  MoveL 8802 to (-24.03, 35.21, 125.68) mm, rotated rx 180 ry 0 rz 180 deg; joints [-34.794, -28.488, 103.329, 69.378, 37.567, -64.603]
  MoveL 8803 to (-24.03, 35.21, 125.68) mm, rotated rx 180 ry 0 rz 180 deg; joints [-34.794, -28.488, 103.329, 69.378, 37.567, -64.603]
  Call Extruder(470.65922)
  MoveL 8804 to (-23.64, 35.16, 125.68) mm, rotated rx 180 ry 0 rz 180 deg; joints [-34.738, -28.447, 103.308, 69.362, 37.51, -64.602]
  MoveL 8805 to (-23.64, 35.16, 125.68) mm, rotated rx 180 ry 0 rz 180 deg; joints [-34.738, -28.447, 103.308, 69.362, 37.51, -64.602]
  Call Extruder(470.90490)
  MoveL 8806 to (-23.15, 35.11, 125.68) mm, rotated rx 180 ry 0 rz 180 deg; joints [-34.671, -28.395, 103.28, 69.345, 37.441, -64.602]
  MoveL 8807 to (-23.15, 35.11, 125.68) mm, rotated rx 180 ry 0 rz 180 deg; joints [-34.671, -28.395, 103.28, 69.345, 37.441, -64.602]
  Call Extruder(471.19963)
  MoveL 8808 to (-22.56, 35.07, 125.68) mm, rotated rx 180 ry 0 rz 180 deg; joints [-34.592, -28.331, 103.247, 69.326, 37.359, -64.604]
  MoveL 8809 to (-22.56, 35.07, 125.68) mm, rotated rx 180 ry 0 rz 180 deg; joints [-34.592, -28.331, 103.247, 69.326, 37.359, -64.604]
  Call Extruder(471.49303)
  MoveL 8810 to (-21.97, 35.02, 125.68) mm, rotated rx -180 ry 0 rz 180 deg; joints [-34.512, -28.267, 103.213, 69.307, 37.276, -64.606]
  MoveL 8811 to (-21.97, 35.02, 125.68) mm, rotated rx -180 ry 0 rz 180 deg; joints [-34.512, -28.267, 103.213, 69.307, 37.276, -64.606]
  Call Extruder(471.92636)
  MoveL 8812 to (-21.1, 34.98, 125.68) mm, rotated rx 180 ry 0 rz -180 deg; joints [-34.399, -28.17, 103.162, 69.282, 37.158, -64.612]
  MoveL 8813 to (-21.1, 34.98, 125.68) mm, rotated rx 180 ry 0 rz -180 deg; joints [-34.399, -28.17, 103.162, 69.282, 37.158, -64.612]
  Call Extruder(472.49852)
  MoveL 8814 to (-19.94, 34.93, 125.68) mm, rotated rx 180 ry 0 rz 180 deg; joints [-34.253, -28.04, 103.092, 69.254, 37.004, -64.624]
  MoveL 8815 to (-19.94, 34.93, 125.68) mm, rotated rx 180 ry 0 rz 180 deg; joints [-34.253, -28.04, 103.092, 69.254, 37.004, -64.624]
  Call Extruder(472.92635)
  MoveL 8816 to (-19.06, 34.91, 125.68) mm, rotated rx -180 ry 0 rz 180 deg; joints [-34.146, -27.941, 103.039, 69.235, 36.891, -64.635]
  Call Extruder(589.57504)
  MoveL 8817 to (219.06, 34.91, 125.68) mm, rotated rx 180 ry 0 rz 180 deg; joints [-18.248, 4.075, 77.332, 65.623, 20.108, -64.241]
  MoveL 8818 to (219.06, 34.91, 125.68) mm, rotated rx 180 ry 0 rz 180 deg; joints [-18.248, 4.075, 77.332, 65.623, 20.108, -64.241]
  Call Extruder(590.29061)
  MoveL 8819 to (220.52, 34.95, 125.68) mm, rotated rx -180 ry 0 rz 180 deg; joints [-18.199, 4.301, 77.091, 65.523, 20.07, -64.141]
  MoveL 8820 to (220.52, 34.95, 125.68) mm, rotated rx -180 ry 0 rz 180 deg; joints [-18.199, 4.301, 77.091, 65.523, 20.07, -64.141]
  Call Extruder(590.86535)
  MoveL 8821 to (221.68, 35, 125.68) mm, rotated rx 180 ry 0 rz 180 deg; joints [-18.162, 4.483, 76.896, 65.442, 20.042, -64.062]
  MoveL 8822 to (221.68, 35, 125.68) mm, rotated rx 180 ry 0 rz 180 deg; joints [-18.162, 4.483, 76.896, 65.442, 20.042, -64.062]
  Call Extruder(591.15874)
  MoveL 8823 to (222.27, 35.04, 125.68) mm, rotated rx -180 ry 0 rz 180 deg; joints [-18.146, 4.576, 76.796, 65.404, 20.03, -64.024]
  MoveL 8824 to (222.27, 35.04, 125.68) mm, rotated rx -180 ry 0 rz 180 deg; joints [-18.146, 4.576, 76.796, 65.404, 20.03, -64.024]
  Call Extruder(591.45347)
  MoveL 8825 to (222.86, 35.09, 125.68) mm, rotated rx 180 ry 0 rz 180 deg; joints [-18.13, 4.669, 76.695, 65.366, 20.018, -63.986]
  MoveL 8826 to (222.86, 35.09, 125.68) mm, rotated rx 180 ry 0 rz 180 deg; joints [-18.13, 4.669, 76.695, 65.366, 20.018, -63.986]
  Call Extruder(591.74952)
  MoveL 8827 to (223.45, 35.14, 125.68) mm, rotated rx 180 ry 0 rz -180 deg; joints [-18.113, 4.763, 76.594, 65.327, 20.007, -63.947]
  MoveL 8828 to (223.45, 35.14, 125.68) mm, rotated rx 180 ry 0 rz -180 deg; joints [-18.113, 4.763, 76.594, 65.327, 20.007, -63.947]
  Call Extruder(591.94580)
  MoveL 8829 to (223.84, 35.18, 125.68) mm, rotated rx -180 ry 0 rz 180 deg; joints [-18.104, 4.825, 76.527, 65.303, 20.001, -63.923]
  MoveL 8830 to (223.84, 35.18, 125.68) mm, rotated rx -180 ry 0 rz 180 deg; joints [-18.104, 4.825, 76.527, 65.303, 20.001, -63.923]
  Call Extruder(592.14294)
  MoveL 8831 to (224.22, 35.23, 125.68) mm, rotated rx -180 ry 0 rz 180 deg; joints [-18.095, 4.888, 76.46, 65.279, 19.995, -63.899]
  MoveL 8832 to (224.22, 35.23, 125.68) mm, rotated rx -180 ry 0 rz 180 deg; joints [-18.095, 4.888, 76.46, 65.279, 19.995, -63.899]
  Call Extruder(592.34095)
  MoveL 8833 to (224.61, 35.27, 125.68) mm, rotated rx 180 ry 0 rz 180 deg; joints [-18.087, 4.95, 76.393, 65.255, 19.989, -63.875]
  MoveL 8834 to (224.61, 35.27, 125.68) mm, rotated rx 180 ry 0 rz 180 deg; joints [-18.087, 4.95, 76.393, 65.255, 19.989, -63.875]
  Call Extruder(592.53982)
  MoveL 8835 to (225, 35.32, 125.68) mm, rotated rx 180 ry 0 rz 180 deg; joints [-18.078, 5.012, 76.325, 65.231, 19.983, -63.85]
  MoveL 8836 to (225, 35.32, 125.68) mm, rotated rx 180 ry 0 rz 180 deg; joints [-18.078, 5.012, 76.325, 65.231, 19.983, -63.85]
  Call Extruder(592.71890)
  MoveL 8837 to (225.34, 35.37, 125.68) mm, rotated rx 180 ry 0 rz 180 deg; joints [-18.07, 5.068, 76.264, 65.21, 19.979, -63.829]
  MoveL 8838 to (225.34, 35.37, 125.68) mm, rotated rx 180 ry 0 rz 180 deg; joints [-18.07, 5.068, 76.264, 65.21, 19.979, -63.829]
  Call Extruder(592.87809)
  MoveL 8839 to (225.65, 35.42, 125.68) mm, rotated rx 180 ry 0 rz 180 deg; joints [-18.065, 5.118, 76.21, 65.192, 19.975, -63.811]
  MoveL 8840 to (225.65, 35.42, 125.68) mm, rotated rx 180 ry 0 rz 180 deg; joints [-18.065, 5.118, 76.21, 65.192, 19.975, -63.811]
  Call Extruder(593.03800)
  MoveL 8841 to (225.96, 35.46, 125.68) mm, rotated rx 180 ry 0 rz 180 deg; joints [-18.059, 5.168, 76.156, 65.174, 19.972, -63.793]
  MoveL 8842 to (225.96, 35.46, 125.68) mm, rotated rx 180 ry 0 rz 180 deg; joints [-18.059, 5.168, 76.156, 65.174, 19.972, -63.793]
  Call Extruder(593.19864)
  MoveL 8843 to (226.26, 35.51, 125.68) mm, rotated rx 180 ry 0 rz 180 deg; joints [-18.054, 5.218, 76.102, 65.156, 19.969, -63.775]
  MoveL 8844 to (226.26, 35.51, 125.68) mm, rotated rx 180 ry 0 rz 180 deg; joints [-18.054, 5.218, 76.102, 65.156, 19.969, -63.775]
  Call Extruder(593.36001)
  MoveL 8845 to (226.57, 35.56, 125.68) mm, rotated rx -180 ry 0 rz 180 deg; joints [-18.048, 5.268, 76.048, 65.138, 19.966, -63.757]
  MoveL 8846 to (226.57, 35.56, 125.68) mm, rotated rx -180 ry 0 rz 180 deg; joints [-18.048, 5.268, 76.048, 65.138, 19.966, -63.757]
  Call Extruder(593.52210)
  MoveL 8847 to (226.87, 35.61, 125.68) mm, rotated rx 180 ry 0 rz -180 deg; joints [-18.042, 5.318, 75.993, 65.12, 19.962, -63.738]
  MoveL 8848 to (226.87, 35.61, 125.68) mm, rotated rx 180 ry 0 rz -180 deg; joints [-18.042, 5.318, 75.993, 65.12, 19.962, -63.738]
  Call Extruder(593.67030)
  MoveL 8849 to (227.15, 35.66, 125.68) mm, rotated rx 180 ry 0 rz 180 deg; joints [-18.038, 5.364, 75.944, 65.104, 19.96, -63.722]
  MoveL 8850 to (227.15, 35.66, 125.68) mm, rotated rx 180 ry 0 rz 180 deg; joints [-18.038, 5.364, 75.944, 65.104, 19.96, -63.722]
  Call Extruder(593.80453)
  MoveL 8851 to (227.4, 35.71, 125.68) mm, rotated rx 180 ry 0 rz 180 deg; joints [-18.034, 5.405, 75.899, 65.091, 19.958, -63.708]
  MoveL 8852 to (227.4, 35.71, 125.68) mm, rotated rx 180 ry 0 rz 180 deg; joints [-18.034, 5.405, 75.899, 65.091, 19.958, -63.708]
  Call Extruder(593.93938)
  MoveL 8853 to (227.65, 35.76, 125.68) mm, rotated rx 180 ry 0 rz 180 deg; joints [-18.031, 5.446, 75.854, 65.077, 19.957, -63.694]
  MoveL 8854 to (227.65, 35.76, 125.68) mm, rotated rx 180 ry 0 rz 180 deg; joints [-18.031, 5.446, 75.854, 65.077, 19.957, -63.694]
  Call Extruder(594.07483)
  MoveL 8855 to (227.9, 35.81, 125.68) mm, rotated rx 180 ry 0 rz 180 deg; joints [-18.027, 5.488, 75.809, 65.063, 19.955, -63.68]
  MoveL 8856 to (227.9, 35.81, 125.68) mm, rotated rx 180 ry 0 rz 180 deg; joints [-18.027, 5.488, 75.809, 65.063, 19.955, -63.68]
  Call Extruder(594.21089)
  MoveL 8857 to (228.15, 35.86, 125.68) mm, rotated rx 180 ry 0 rz -180 deg; joints [-18.024, 5.529, 75.764, 65.049, 19.954, -63.666]
  MoveL 8858 to (228.15, 35.86, 125.68) mm, rotated rx 180 ry 0 rz -180 deg; joints [-18.024, 5.529, 75.764, 65.049, 19.954, -63.666]
  Call Extruder(594.34757)
  MoveL 8859 to (228.4, 35.91, 125.68) mm, rotated rx 180 ry 0 rz 180 deg; joints [-18.02, 5.57, 75.719, 65.035, 19.952, -63.651]
  MoveL 8860 to (228.4, 35.91, 125.68) mm, rotated rx 180 ry 0 rz 180 deg; joints [-18.02, 5.57, 75.719, 65.035, 19.952, -63.651]
  Call Extruder(594.48485)
  MoveL 8861 to (228.65, 35.96, 125.68) mm, rotated rx 180 ry 0 rz 180 deg; joints [-18.017, 5.612, 75.673, 65.021, 19.951, -63.637]
  MoveL 8862 to (228.65, 35.96, 125.68) mm, rotated rx 180 ry 0 rz 180 deg; joints [-18.017, 5.612, 75.673, 65.021, 19.951, -63.637]
  Call Extruder(594.61052)
  MoveL 8863 to (228.87, 36, 125.68) mm, rotated rx 180 ry 0 rz 180 deg; joints [-18.014, 5.649, 75.632, 65.009, 19.95, -63.624]
  MoveL 8864 to (228.87, 36, 125.68) mm, rotated rx 180 ry 0 rz 180 deg; joints [-18.014, 5.649, 75.632, 65.009, 19.95, -63.624]
  Call Extruder(594.72447)
  MoveL 8865 to (229.08, 36.05, 125.68) mm, rotated rx -180 ry 0 rz -180 deg; joints [-18.012, 5.684, 75.595, 64.998, 19.949, -63.613]
  MoveL 8866 to (229.08, 36.05, 125.68) mm, rotated rx -180 ry 0 rz -180 deg; joints [-18.012, 5.684, 75.595, 64.998, 19.949, -63.613]
  Call Extruder(594.83887)
  MoveL 8867 to (229.28, 36.09, 125.68) mm, rotated rx 180 ry 0 rz 180 deg; joints [-18.009, 5.718, 75.558, 64.987, 19.948, -63.602]
  MoveL 8868 to (229.28, 36.09, 125.68) mm, rotated rx 180 ry 0 rz 180 deg; joints [-18.009, 5.718, 75.558, 64.987, 19.948, -63.602]
  Call Extruder(594.95372)
  MoveL 8869 to (229.48, 36.14, 125.68) mm, rotated rx -180 ry 0 rz 180 deg; joints [-18.007, 5.752, 75.52, 64.976, 19.947, -63.59]
  MoveL 8870 to (229.48, 36.14, 125.68) mm, rotated rx -180 ry 0 rz 180 deg; joints [-18.007, 5.752, 75.52, 64.976, 19.947, -63.59]
  Call Extruder(595.06902)
  MoveL 8871 to (229.69, 36.18, 125.68) mm, rotated rx 180 ry 0 rz 180 deg; joints [-18.005, 5.786, 75.483, 64.965, 19.947, -63.579]
  MoveL 8872 to (229.69, 36.18, 125.68) mm, rotated rx 180 ry 0 rz 180 deg; joints [-18.005, 5.786, 75.483, 64.965, 19.947, -63.579]
  Call Extruder(595.20041)
  MoveL 8873 to (229.92, 36.25, 125.68) mm, rotated rx 180 ry 0 rz -180 deg; joints [-18.004, 5.825, 75.44, 64.954, 19.947, -63.568]
  MoveL 8874 to (229.92, 36.25, 125.68) mm, rotated rx 180 ry 0 rz -180 deg; joints [-18.004, 5.825, 75.44, 64.954, 19.947, -63.568]
  Call Extruder(595.31352)
  MoveL 8875 to (230.11, 36.31, 125.68) mm, rotated rx 180 ry 0 rz 180 deg; joints [-18.003, 5.858, 75.403, 64.945, 19.948, -63.558]
  MoveL 8876 to (230.11, 36.31, 125.68) mm, rotated rx 180 ry 0 rz 180 deg; joints [-18.003, 5.858, 75.403, 64.945, 19.948, -63.558]
  Call Extruder(595.42707)
  MoveL 8877 to (230.31, 36.37, 125.68) mm, rotated rx 180 ry 0 rz 180 deg; joints [-18.003, 5.892, 75.367, 64.937, 19.949, -63.549]
  MoveL 8878 to (230.31, 36.37, 125.68) mm, rotated rx 180 ry 0 rz 180 deg; joints [-18.003, 5.892, 75.367, 64.937, 19.949, -63.549]
  Call Extruder(595.54106)
  MoveL 8879 to (230.5, 36.43, 125.68) mm, rotated rx 180 ry 0 rz -180 deg; joints [-18.002, 5.925, 75.33, 64.928, 19.95, -63.54]
  MoveL 8880 to (230.5, 36.43, 125.68) mm, rotated rx 180 ry 0 rz -180 deg; joints [-18.002, 5.925, 75.33, 64.928, 19.95, -63.54]
  Call Extruder(595.65549)
  MoveL 8881 to (230.69, 36.49, 125.68) mm, rotated rx 180 ry 0 rz 180 deg; joints [-18.002, 5.959, 75.293, 64.92, 19.951, -63.531]
  MoveL 8882 to (230.69, 36.49, 125.68) mm, rotated rx 180 ry 0 rz 180 deg; joints [-18.002, 5.959, 75.293, 64.92, 19.951, -63.531]
  Call Extruder(595.76739)
  MoveL 8883 to (230.88, 36.55, 125.68) mm, rotated rx 180 ry 0 rz 180 deg; joints [-18.002, 5.991, 75.257, 64.912, 19.953, -63.523]
  MoveL 8884 to (230.88, 36.55, 125.68) mm, rotated rx 180 ry 0 rz 180 deg; joints [-18.002, 5.991, 75.257, 64.912, 19.953, -63.523]
  Call Extruder(595.87973)
  MoveL 8885 to (231.07, 36.61, 125.68) mm, rotated rx 180 ry 0 rz 180 deg; joints [-18.002, 6.024, 75.222, 64.903, 19.954, -63.514]
  MoveL 8886 to (231.07, 36.61, 125.68) mm, rotated rx 180 ry 0 rz 180 deg; joints [-18.002, 6.024, 75.222, 64.903, 19.954, -63.514]
  Call Extruder(595.99252)
  MoveL 8887 to (231.26, 36.67, 125.68) mm, rotated rx 180 ry 0 rz 180 deg; joints [-18.002, 6.057, 75.186, 64.895, 19.956, -63.506]
  MoveL 8888 to (231.26, 36.67, 125.68) mm, rotated rx 180 ry 0 rz 180 deg; joints [-18.002, 6.057, 75.186, 64.895, 19.956, -63.506]
  Call Extruder(596.10575)
  MoveL 8889 to (231.45, 36.73, 125.68) mm, rotated rx 180 ry 0 rz 180 deg; joints [-18.002, 6.089, 75.15, 64.887, 19.957, -63.497]
  MoveL 8890 to (231.45, 36.73, 125.68) mm, rotated rx 180 ry 0 rz 180 deg; joints [-18.002, 6.089, 75.15, 64.887, 19.957, -63.497]
  Call Extruder(596.21943)
  MoveL 8891 to (231.64, 36.79, 125.68) mm, rotated rx 180 ry 0 rz 180 deg; joints [-18.002, 6.122, 75.114, 64.879, 19.958, -63.488]
  MoveL 8892 to (231.64, 36.79, 125.68) mm, rotated rx 180 ry 0 rz 180 deg; joints [-18.002, 6.122, 75.114, 64.879, 19.958, -63.488]
  Call Extruder(596.40139)
  MoveL 8893 to (231.93, 36.91, 125.68) mm, rotated rx 180 ry 0 rz 180 deg; joints [-18.005, 6.174, 75.057, 64.87, 19.963, -63.478]
  MoveL 8894 to (231.93, 36.91, 125.68) mm, rotated rx 180 ry 0 rz 180 deg; joints [-18.005, 6.174, 75.057, 64.87, 19.963, -63.478]
  Call Extruder(596.58411)
  MoveL 8895 to (232.22, 37.04, 125.68) mm, rotated rx 180 ry 0 rz -180 deg; joints [-18.008, 6.226, 74.999, 64.86, 19.968, -63.467]
  MoveL 8896 to (232.22, 37.04, 125.68) mm, rotated rx 180 ry 0 rz -180 deg; joints [-18.008, 6.226, 74.999, 64.86, 19.968, -63.467]
  Call Extruder(596.75452)
  MoveL 8897 to (232.49, 37.15, 125.68) mm, rotated rx 180 ry 0 rz 180 deg; joints [-18.011, 6.274, 74.946, 64.852, 19.973, -63.458]
  MoveL 8898 to (232.49, 37.15, 125.68) mm, rotated rx 180 ry 0 rz 180 deg; joints [-18.011, 6.274, 74.946, 64.852, 19.973, -63.458]
  Call Extruder(596.91252)
  MoveL 8899 to (232.74, 37.26, 125.68) mm, rotated rx -180 ry 0 rz -180 deg; joints [-18.013, 6.319, 74.897, 64.844, 19.977, -63.449]
  MoveL 8900 to (232.74, 37.26, 125.68) mm, rotated rx -180 ry 0 rz -180 deg; joints [-18.013, 6.319, 74.897, 64.844, 19.977, -63.449]
  Call Extruder(597.07112)
  MoveL 8901 to (232.99, 37.36, 125.68) mm, rotated rx -180 ry 0 rz 180 deg; joints [-18.016, 6.363, 74.848, 64.836, 19.982, -63.44]
  MoveL 8902 to (232.99, 37.36, 125.68) mm, rotated rx -180 ry 0 rz 180 deg; joints [-18.016, 6.363, 74.848, 64.836, 19.982, -63.44]
  Call Extruder(597.27729)
  MoveL 8903 to (233.29, 37.54, 125.68) mm, rotated rx 180 ry 0 rz 180 deg; joints [-18.024, 6.42, 74.785, 64.832, 19.991, -63.434]
  MoveL 8904 to (233.29, 37.54, 125.68) mm, rotated rx 180 ry 0 rz 180 deg; joints [-18.024, 6.42, 74.785, 64.832, 19.991, -63.434]
  Call Extruder(597.48423)
  MoveL 8905 to (233.6, 37.71, 125.68) mm, rotated rx 180 ry 0 rz 180 deg; joints [-18.033, 6.477, 74.722, 64.828, 20.001, -63.429]
  MoveL 8906 to (233.6, 37.71, 125.68) mm, rotated rx 180 ry 0 rz 180 deg; joints [-18.033, 6.477, 74.722, 64.828, 20.001, -63.429]
  Call Extruder(597.69196)
  MoveL 8907 to (233.9, 37.89, 125.68) mm, rotated rx -180 ry 0 rz -180 deg; joints [-18.041, 6.534, 74.66, 64.823, 20.011, -63.423]
  MoveL 8908 to (233.9, 37.89, 125.68) mm, rotated rx -180 ry 0 rz -180 deg; joints [-18.041, 6.534, 74.66, 64.823, 20.011, -63.423]
  Call Extruder(597.90046)
  MoveL 8909 to (234.21, 38.07, 125.68) mm, rotated rx 180 ry 0 rz 180 deg; joints [-18.049, 6.59, 74.597, 64.819, 20.021, -63.417]
  MoveL 8910 to (234.21, 38.07, 125.68) mm, rotated rx 180 ry 0 rz 180 deg; joints [-18.049, 6.59, 74.597, 64.819, 20.021, -63.417]
  Call Extruder(598.08001)
  MoveL 8911 to (234.45, 38.24, 125.68) mm, rotated rx 180 ry 0 rz 180 deg; joints [-18.06, 6.638, 74.544, 64.82, 20.033, -63.416]
  MoveL 8912 to (234.45, 38.24, 125.68) mm, rotated rx 180 ry 0 rz 180 deg; joints [-18.06, 6.638, 74.544, 64.82, 20.033, -63.416]
  Call Extruder(598.41342)
  MoveL 8913 to (234.9, 38.57, 125.68) mm, rotated rx 180 ry 0 rz 180 deg; joints [-18.079, 6.726, 74.446, 64.821, 20.055, -63.414]
  MoveL 8914 to (234.9, 38.57, 125.68) mm, rotated rx 180 ry 0 rz 180 deg; joints [-18.079, 6.726, 74.446, 64.821, 20.055, -63.414]
  Call Extruder(598.74802)
  MoveL 8915 to (235.35, 38.9, 125.68) mm, rotated rx 180 ry 0 rz 180 deg; joints [-18.099, 6.814, 74.348, 64.823, 20.076, -63.412]
  Call Extruder(599.57597)
  MoveL 8916 to (236.39, 39.81, 125.68) mm, rotated rx 180 ry 0 rz -180 deg; joints [-18.16, 7.025, 74.114, 64.844, 20.142, -63.425]
  Call Extruder(600.40391)
  MoveL 8917 to (237.3, 40.85, 125.68) mm, rotated rx 180 ry 0 rz -180 deg; joints [-18.24, 7.223, 73.892, 64.889, 20.222, -63.46]
  Call Extruder(600.57121)
  MoveL 8918 to (237.47, 41.07, 125.68) mm, rotated rx -180 ry 0 rz 180 deg; joints [-18.258, 7.26, 73.85, 64.902, 20.241, -63.471]
  MoveL 8919 to (237.47, 41.07, 125.68) mm, rotated rx -180 ry 0 rz 180 deg; joints [-18.258, 7.26, 73.85, 64.902, 20.241, -63.471]
  Call Extruder(600.90463)
  MoveL 8920 to (237.8, 41.52, 125.68) mm, rotated rx 180 ry 0 rz 180 deg; joints [-18.295, 7.336, 73.766, 64.927, 20.277, -63.491]
  MoveL 8921 to (237.8, 41.52, 125.68) mm, rotated rx 180 ry 0 rz 180 deg; joints [-18.295, 7.336, 73.766, 64.927, 20.277, -63.491]
  Call Extruder(601.23686)
  MoveL 8922 to (238.12, 41.98, 125.68) mm, rotated rx -180 ry 0 rz 180 deg; joints [-18.332, 7.412, 73.681, 64.952, 20.314, -63.512]
  MoveL 8923 to (238.12, 41.98, 125.68) mm, rotated rx -180 ry 0 rz 180 deg; joints [-18.332, 7.412, 73.681, 64.952, 20.314, -63.512]
  Call Extruder(601.35455)
  MoveL 8924 to (238.22, 42.15, 125.68) mm, rotated rx 180 ry 0 rz 180 deg; joints [-18.346, 7.436, 73.653, 64.963, 20.329, -63.522]
  MoveL 8925 to (238.22, 42.15, 125.68) mm, rotated rx 180 ry 0 rz 180 deg; joints [-18.346, 7.436, 73.653, 64.963, 20.329, -63.522]
  Call Extruder(601.56228)
  MoveL 8926 to (238.4, 42.45, 125.68) mm, rotated rx 180 ry 0 rz 180 deg; joints [-18.373, 7.48, 73.604, 64.984, 20.354, -63.539]
  MoveL 8927 to (238.4, 42.45, 125.68) mm, rotated rx 180 ry 0 rz 180 deg; joints [-18.373, 7.48, 73.604, 64.984, 20.354, -63.539]
  Call Extruder(601.76922)
  MoveL 8928 to (238.57, 42.75, 125.68) mm, rotated rx 180 ry 0 rz -180 deg; joints [-18.399, 7.524, 73.555, 65.004, 20.38, -63.557]
  MoveL 8929 to (238.57, 42.75, 125.68) mm, rotated rx 180 ry 0 rz -180 deg; joints [-18.399, 7.524, 73.555, 65.004, 20.38, -63.557]
  Call Extruder(601.97539)
  MoveL 8930 to (238.75, 43.06, 125.68) mm, rotated rx 180 ry 0 rz 180 deg; joints [-18.425, 7.568, 73.506, 65.025, 20.406, -63.574]
  MoveL 8931 to (238.75, 43.06, 125.68) mm, rotated rx 180 ry 0 rz 180 deg; joints [-18.425, 7.568, 73.506, 65.025, 20.406, -63.574]
  Call Extruder(602.15708)
  MoveL 8932 to (238.89, 43.34, 125.68) mm, rotated rx 180 ry 0 rz 180 deg; joints [-18.45, 7.605, 73.464, 65.045, 20.43, -63.591]
  MoveL 8933 to (238.89, 43.34, 125.68) mm, rotated rx 180 ry 0 rz 180 deg; joints [-18.45, 7.605, 73.464, 65.045, 20.43, -63.591]
  Call Extruder(602.31509)
  MoveL 8934 to (239, 43.58, 125.68) mm, rotated rx 180 ry 0 rz 180 deg; joints [-18.472, 7.635, 73.43, 65.064, 20.452, -63.608]
  MoveL 8935 to (239, 43.58, 125.68) mm, rotated rx 180 ry 0 rz 180 deg; joints [-18.472, 7.635, 73.43, 65.064, 20.452, -63.608]
  Call Extruder(602.47250)
  MoveL 8936 to (239.11, 43.83, 125.68) mm, rotated rx 180 ry 0 rz 180 deg; joints [-18.495, 7.665, 73.396, 65.084, 20.474, -63.626]
  MoveL 8937 to (239.11, 43.83, 125.68) mm, rotated rx 180 ry 0 rz 180 deg; joints [-18.495, 7.665, 73.396, 65.084, 20.474, -63.626]
  Call Extruder(602.65521)
  MoveL 8938 to (239.23, 44.13, 125.68) mm, rotated rx 180 ry 0 rz 180 deg; joints [-18.522, 7.7, 73.357, 65.107, 20.5, -63.646]
  MoveL 8939 to (239.23, 44.13, 125.68) mm, rotated rx 180 ry 0 rz 180 deg; joints [-18.522, 7.7, 73.357, 65.107, 20.5, -63.646]
  Call Extruder(602.83717)
  MoveL 8940 to (239.35, 44.42, 125.68) mm, rotated rx 180 ry 0 rz 180 deg; joints [-18.549, 7.734, 73.318, 65.131, 20.526, -63.667]
  MoveL 8941 to (239.35, 44.42, 125.68) mm, rotated rx 180 ry 0 rz 180 deg; joints [-18.549, 7.734, 73.318, 65.131, 20.526, -63.667]
  Call Extruder(602.98450)
  MoveL 8942 to (239.44, 44.66, 125.68) mm, rotated rx 180 ry 0 rz -180 deg; joints [-18.571, 7.762, 73.287, 65.15, 20.547, -63.684]
  MoveL 8943 to (239.44, 44.66, 125.68) mm, rotated rx 180 ry 0 rz -180 deg; joints [-18.571, 7.762, 73.287, 65.15, 20.547, -63.684]
  Call Extruder(603.09774)
  MoveL 8944 to (239.5, 44.85, 125.68) mm, rotated rx -180 ry 0 rz 180 deg; joints [-18.589, 7.782, 73.265, 65.167, 20.564, -63.699]
  MoveL 8945 to (239.5, 44.85, 125.68) mm, rotated rx -180 ry 0 rz 180 deg; joints [-18.589, 7.782, 73.265, 65.167, 20.564, -63.699]
  Call Extruder(603.21053)
  MoveL 8946 to (239.56, 45.03, 125.68) mm, rotated rx 180 ry 0 rz 180 deg; joints [-18.607, 7.801, 73.242, 65.183, 20.581, -63.713]
  MoveL 8947 to (239.56, 45.03, 125.68) mm, rotated rx 180 ry 0 rz 180 deg; joints [-18.607, 7.801, 73.242, 65.183, 20.581, -63.713]
  Call Extruder(603.32287)
  MoveL 8948 to (239.62, 45.22, 125.68) mm, rotated rx 180 ry 0 rz 180 deg; joints [-18.625, 7.821, 73.22, 65.2, 20.598, -63.728]
  MoveL 8949 to (239.62, 45.22, 125.68) mm, rotated rx 180 ry 0 rz 180 deg; joints [-18.625, 7.821, 73.22, 65.2, 20.598, -63.728]
  Call Extruder(603.43477)
  MoveL 8950 to (239.68, 45.41, 125.68) mm, rotated rx 180 ry 0 rz -180 deg; joints [-18.642, 7.841, 73.198, 65.216, 20.615, -63.742]
  MoveL 8951 to (239.68, 45.41, 125.68) mm, rotated rx 180 ry 0 rz -180 deg; joints [-18.642, 7.841, 73.198, 65.216, 20.615, -63.742]
  Call Extruder(603.55618)
  MoveL 8952 to (239.75, 45.62, 125.68) mm, rotated rx 180 ry 0 rz -180 deg; joints [-18.662, 7.862, 73.174, 65.234, 20.634, -63.758]
  MoveL 8953 to (239.75, 45.62, 125.68) mm, rotated rx 180 ry 0 rz -180 deg; joints [-18.662, 7.862, 73.174, 65.234, 20.634, -63.758]
  Call Extruder(603.68697)
  MoveL 8954 to (239.81, 45.84, 125.68) mm, rotated rx 180 ry 0 rz 180 deg; joints [-18.683, 7.885, 73.148, 65.253, 20.654, -63.775]
  MoveL 8955 to (239.81, 45.84, 125.68) mm, rotated rx 180 ry 0 rz 180 deg; joints [-18.683, 7.885, 73.148, 65.253, 20.654, -63.775]
  Call Extruder(603.81719)
  MoveL 8956 to (239.88, 46.06, 125.68) mm, rotated rx 180 ry 0 rz -180 deg; joints [-18.705, 7.908, 73.122, 65.273, 20.675, -63.793]
  MoveL 8957 to (239.88, 46.06, 125.68) mm, rotated rx 180 ry 0 rz -180 deg; joints [-18.705, 7.908, 73.122, 65.273, 20.675, -63.793]
  Call Extruder(603.94685)
  MoveL 8958 to (239.95, 46.29, 125.68) mm, rotated rx 180 ry 0 rz 180 deg; joints [-18.726, 7.93, 73.096, 65.292, 20.695, -63.81]
  MoveL 8959 to (239.95, 46.29, 125.68) mm, rotated rx 180 ry 0 rz 180 deg; joints [-18.726, 7.93, 73.096, 65.292, 20.695, -63.81]
  Call Extruder(604.07595)
  MoveL 8960 to (240.02, 46.51, 125.68) mm, rotated rx 180 ry 0 rz -180 deg; joints [-18.747, 7.953, 73.071, 65.312, 20.715, -63.827]
  MoveL 8961 to (240.02, 46.51, 125.68) mm, rotated rx 180 ry 0 rz -180 deg; joints [-18.747, 7.953, 73.071, 65.312, 20.715, -63.827]
  Call Extruder(604.19100)
  MoveL 8962 to (240.06, 46.72, 125.68) mm, rotated rx 180 ry 0 rz 180 deg; joints [-18.767, 7.971, 73.05, 65.331, 20.734, -63.844]
  MoveL 8963 to (240.06, 46.72, 125.68) mm, rotated rx 180 ry 0 rz 180 deg; joints [-18.767, 7.971, 73.05, 65.331, 20.734, -63.844]
  Call Extruder(604.30560)
  MoveL 8964 to (240.11, 46.92, 125.68) mm, rotated rx 180 ry 0 rz 180 deg; joints [-18.787, 7.989, 73.03, 65.35, 20.753, -63.862]
  MoveL 8965 to (240.11, 46.92, 125.68) mm, rotated rx 180 ry 0 rz 180 deg; joints [-18.787, 7.989, 73.03, 65.35, 20.753, -63.862]
  Call Extruder(604.41975)
  MoveL 8966 to (240.15, 47.12, 125.68) mm, rotated rx 180 ry 0 rz 180 deg; joints [-18.807, 8.007, 73.009, 65.37, 20.772, -63.879]
  MoveL 8967 to (240.15, 47.12, 125.68) mm, rotated rx 180 ry 0 rz 180 deg; joints [-18.807, 8.007, 73.009, 65.37, 20.772, -63.879]
  Call Extruder(604.53345)
  MoveL 8968 to (240.2, 47.33, 125.68) mm, rotated rx -180 ry 0 rz 180 deg; joints [-18.827, 8.026, 72.989, 65.389, 20.791, -63.896]
  MoveL 8969 to (240.2, 47.33, 125.68) mm, rotated rx -180 ry 0 rz 180 deg; joints [-18.827, 8.026, 72.989, 65.389, 20.791, -63.896]
  Call Extruder(604.65886)
  MoveL 8970 to (240.24, 47.56, 125.68) mm, rotated rx 180 ry 0 rz 180 deg; joints [-18.85, 8.045, 72.966, 65.41, 20.812, -63.915]
  MoveL 8971 to (240.24, 47.56, 125.68) mm, rotated rx 180 ry 0 rz 180 deg; joints [-18.85, 8.045, 72.966, 65.41, 20.812, -63.915]
  Call Extruder(604.79583)
  MoveL 8972 to (240.29, 47.8, 125.68) mm, rotated rx 180 ry 0 rz 180 deg; joints [-18.874, 8.067, 72.942, 65.434, 20.836, -63.936]
  MoveL 8973 to (240.29, 47.8, 125.68) mm, rotated rx 180 ry 0 rz 180 deg; joints [-18.874, 8.067, 72.942, 65.434, 20.836, -63.936]
  Call Extruder(604.93220)
  MoveL 8974 to (240.34, 48.05, 125.68) mm, rotated rx 180 ry 0 rz 180 deg; joints [-18.899, 8.088, 72.918, 65.457, 20.859, -63.957]
  MoveL 8975 to (240.34, 48.05, 125.68) mm, rotated rx 180 ry 0 rz 180 deg; joints [-18.899, 8.088, 72.918, 65.457, 20.859, -63.957]
  Call Extruder(605.06796)
  MoveL 8976 to (240.39, 48.3, 125.68) mm, rotated rx 180 ry 0 rz 180 deg; joints [-18.923, 8.11, 72.893, 65.481, 20.882, -63.978]
  MoveL 8977 to (240.39, 48.3, 125.68) mm, rotated rx 180 ry 0 rz 180 deg; joints [-18.923, 8.11, 72.893, 65.481, 20.882, -63.978]
  Call Extruder(605.20311)
  MoveL 8978 to (240.44, 48.55, 125.68) mm, rotated rx 180 ry 0 rz 180 deg; joints [-18.948, 8.131, 72.869, 65.504, 20.906, -63.999]
  MoveL 8979 to (240.44, 48.55, 125.68) mm, rotated rx 180 ry 0 rz 180 deg; joints [-18.948, 8.131, 72.869, 65.504, 20.906, -63.999]
  Call Extruder(605.33764)
  MoveL 8980 to (240.49, 48.8, 125.68) mm, rotated rx 180 ry 0 rz 180 deg; joints [-18.973, 8.153, 72.845, 65.527, 20.929, -64.02]
  MoveL 8981 to (240.49, 48.8, 125.68) mm, rotated rx 180 ry 0 rz 180 deg; joints [-18.973, 8.153, 72.845, 65.527, 20.929, -64.02]
  Call Extruder(605.47157)
  MoveL 8982 to (240.54, 49.05, 125.68) mm, rotated rx -180 ry 0 rz 180 deg; joints [-18.997, 8.174, 72.821, 65.55, 20.952, -64.041]
  MoveL 8983 to (240.54, 49.05, 125.68) mm, rotated rx -180 ry 0 rz 180 deg; joints [-18.997, 8.174, 72.821, 65.55, 20.952, -64.041]
  Call Extruder(605.61944)
  MoveL 8984 to (240.59, 49.33, 125.68) mm, rotated rx 180 ry 0 rz 180 deg; joints [-19.025, 8.197, 72.794, 65.577, 20.978, -64.064]
  MoveL 8985 to (240.59, 49.33, 125.68) mm, rotated rx 180 ry 0 rz 180 deg; joints [-19.025, 8.197, 72.794, 65.577, 20.978, -64.064]
  Call Extruder(605.78118)
  MoveL 8986 to (240.64, 49.63, 125.68) mm, rotated rx 180 ry 0 rz 180 deg; joints [-19.055, 8.222, 72.767, 65.606, 21.007, -64.091]
  MoveL 8987 to (240.64, 49.63, 125.68) mm, rotated rx 180 ry 0 rz 180 deg; joints [-19.055, 8.222, 72.767, 65.606, 21.007, -64.091]
  Call Extruder(605.94220)
  MoveL 8988 to (240.69, 49.94, 125.68) mm, rotated rx 180 ry 0 rz 180 deg; joints [-19.086, 8.246, 72.739, 65.635, 21.036, -64.117]
  MoveL 8989 to (240.69, 49.94, 125.68) mm, rotated rx 180 ry 0 rz 180 deg; joints [-19.086, 8.246, 72.739, 65.635, 21.036, -64.117]
  Call Extruder(606.10249)
  MoveL 8990 to (240.74, 50.24, 125.68) mm, rotated rx 180 ry 0 rz 180 deg; joints [-19.116, 8.271, 72.711, 65.664, 21.064, -64.143]
  MoveL 8991 to (240.74, 50.24, 125.68) mm, rotated rx 180 ry 0 rz 180 deg; joints [-19.116, 8.271, 72.711, 65.664, 21.064, -64.143]
  Call Extruder(606.26205)
  MoveL 8992 to (240.78, 50.55, 125.68) mm, rotated rx 180 ry 0 rz 180 deg; joints [-19.146, 8.295, 72.683, 65.693, 21.093, -64.169]
  MoveL 8993 to (240.78, 50.55, 125.68) mm, rotated rx 180 ry 0 rz 180 deg; joints [-19.146, 8.295, 72.683, 65.693, 21.093, -64.169]
  Call Extruder(606.42088)
  MoveL 8994 to (240.83, 50.86, 125.68) mm, rotated rx 180 ry 0 rz 180 deg; joints [-19.177, 8.32, 72.655, 65.722, 21.122, -64.195]
  MoveL 8995 to (240.83, 50.86, 125.68) mm, rotated rx 180 ry 0 rz 180 deg; joints [-19.177, 8.32, 72.655, 65.722, 21.122, -64.195]
  Call Extruder(606.59956)
  MoveL 8996 to (240.88, 51.2, 125.68) mm, rotated rx 180 ry 0 rz 180 deg; joints [-19.212, 8.346, 72.625, 65.756, 21.155, -64.224]
  MoveL 8997 to (240.88, 51.2, 125.68) mm, rotated rx 180 ry 0 rz 180 deg; joints [-19.212, 8.346, 72.625, 65.756, 21.155, -64.224]
  Call Extruder(606.79800)
  MoveL 8998 to (240.92, 51.59, 125.68) mm, rotated rx -180 ry 0 rz 180 deg; joints [-19.251, 8.375, 72.592, 65.793, 21.192, -64.258]
  MoveL 8999 to (240.92, 51.59, 125.68) mm, rotated rx -180 ry 0 rz 180 deg; joints [-19.251, 8.375, 72.592, 65.793, 21.192, -64.258]
  Call Extruder(606.99557)
  MoveL 9000 to (240.97, 51.98, 125.68) mm, rotated rx 180 ry 0 rz 180 deg; joints [-19.29, 8.404, 72.559, 65.831, 21.228, -64.292]
  MoveL 9001 to (240.97, 51.98, 125.68) mm, rotated rx 180 ry 0 rz 180 deg; joints [-19.29, 8.404, 72.559, 65.831, 21.228, -64.292]
  Call Extruder(607.19228)
  MoveL 9002 to (241.02, 52.36, 125.68) mm, rotated rx 180 ry 0 rz 180 deg; joints [-19.329, 8.433, 72.526, 65.868, 21.265, -64.325]
  MoveL 9003 to (241.02, 52.36, 125.68) mm, rotated rx 180 ry 0 rz 180 deg; joints [-19.329, 8.433, 72.526, 65.868, 21.265, -64.325]
  Call Extruder(607.38812)
  MoveL 9004 to (241.06, 52.75, 125.68) mm, rotated rx 180 ry 0 rz 180 deg; joints [-19.368, 8.462, 72.493, 65.905, 21.302, -64.359]
  MoveL 9005 to (241.06, 52.75, 125.68) mm, rotated rx 180 ry 0 rz 180 deg; joints [-19.368, 8.462, 72.493, 65.905, 21.302, -64.359]
  Call Extruder(607.68356)
  MoveL 9006 to (241.11, 53.34, 125.68) mm, rotated rx 180 ry 0 rz 180 deg; joints [-19.428, 8.502, 72.447, 65.964, 21.359, -64.411]
  MoveL 9007 to (241.11, 53.34, 125.68) mm, rotated rx 180 ry 0 rz 180 deg; joints [-19.428, 8.502, 72.447, 65.964, 21.359, -64.411]
  Call Extruder(607.97766)
  MoveL 9008 to (241.15, 53.93, 125.68) mm, rotated rx 180 ry 0 rz 180 deg; joints [-19.488, 8.543, 72.401, 66.022, 21.415, -64.463]
  MoveL 9009 to (241.15, 53.93, 125.68) mm, rotated rx 180 ry 0 rz 180 deg; joints [-19.488, 8.543, 72.401, 66.022, 21.415, -64.463]
  Call Extruder(608.27044)
  MoveL 9010 to (241.2, 54.52, 125.68) mm, rotated rx -180 ry 0 rz 180 deg; joints [-19.548, 8.584, 72.355, 66.079, 21.472, -64.515]
  MoveL 9011 to (241.2, 54.52, 125.68) mm, rotated rx -180 ry 0 rz 180 deg; joints [-19.548, 8.584, 72.355, 66.079, 21.472, -64.515]
  Call Extruder(608.84389)
  MoveL 9012 to (241.25, 55.68, 125.68) mm, rotated rx 180 ry 0 rz 180 deg; joints [-19.668, 8.657, 72.271, 66.195, 21.584, -64.62]
  MoveL 9013 to (241.25, 55.68, 125.68) mm, rotated rx 180 ry 0 rz 180 deg; joints [-19.668, 8.657, 72.271, 66.195, 21.584, -64.62]
  Call Extruder(609.55772)
  MoveL 9014 to (241.29, 57.14, 125.68) mm, rotated rx 180 ry 0 rz 180 deg; joints [-19.819, 8.746, 72.169, 66.34, 21.726, -64.75]
  Call Extruder(651.62260)
  MoveL 9015 to (241.29, 142.86, 125.68) mm, rotated rx 180 ry 0 rz 180 deg; joints [-28.232, 14.886, 64.835, 71.616, 29.9, -69.024]
  Call Extruder(652.05103)
  MoveL 9016 to (241.27, 143.74, 125.68) mm, rotated rx -180 ry 0 rz -180 deg; joints [-28.313, 14.959, 64.744, 71.644, 29.981, -69.04]
  MoveL 9017 to (241.27, 143.74, 125.68) mm, rotated rx -180 ry 0 rz -180 deg; joints [-28.313, 14.959, 64.744, 71.644, 29.981, -69.04]
  Call Extruder(652.62448)
  MoveL 9018 to (241.22, 144.9, 125.68) mm, rotated rx 180 ry 0 rz 180 deg; joints [-28.421, 15.053, 64.627, 71.683, 30.089, -69.063]
  MoveL 9019 to (241.22, 144.9, 125.68) mm, rotated rx 180 ry 0 rz 180 deg; joints [-28.421, 15.053, 64.627, 71.683, 30.089, -69.063]
  Call Extruder(653.05882)
  MoveL 9020 to (241.18, 145.77, 125.68) mm, rotated rx 180 ry 0 rz 180 deg; joints [-28.503, 15.122, 64.541, 71.714, 30.172, -69.081]
  MoveL 9021 to (241.18, 145.77, 125.68) mm, rotated rx 180 ry 0 rz 180 deg; joints [-28.503, 15.122, 64.541, 71.714, 30.172, -69.081]
  Call Extruder(653.35293)
  MoveL 9022 to (241.13, 146.36, 125.68) mm, rotated rx 180 ry 0 rz -180 deg; joints [-28.559, 15.166, 64.486, 71.736, 30.227, -69.095]
  MoveL 9023 to (241.13, 146.36, 125.68) mm, rotated rx 180 ry 0 rz -180 deg; joints [-28.559, 15.166, 64.486, 71.736, 30.227, -69.095]
  Call Extruder(653.64837)
  MoveL 9024 to (241.09, 146.95, 125.68) mm, rotated rx 180 ry 0 rz 180 deg; joints [-28.615, 15.21, 64.43, 71.757, 30.283, -69.108]
  MoveL 9025 to (241.09, 146.95, 125.68) mm, rotated rx 180 ry 0 rz 180 deg; joints [-28.615, 15.21, 64.43, 71.757, 30.283, -69.108]
  Call Extruder(653.89462)
  MoveL 9026 to (241.04, 147.44, 125.68) mm, rotated rx 180 ry 0 rz 180 deg; joints [-28.662, 15.246, 64.386, 71.776, 30.329, -69.12]
  MoveL 9027 to (241.04, 147.44, 125.68) mm, rotated rx 180 ry 0 rz 180 deg; joints [-28.662, 15.246, 64.386, 71.776, 30.329, -69.12]
  Call Extruder(654.09133)
  MoveL 9028 to (240.99, 147.83, 125.68) mm, rotated rx 180 ry 0 rz 180 deg; joints [-28.7, 15.273, 64.352, 71.791, 30.367, -69.13]
  MoveL 9029 to (240.99, 147.83, 125.68) mm, rotated rx 180 ry 0 rz 180 deg; joints [-28.7, 15.273, 64.352, 71.791, 30.367, -69.13]
  Call Extruder(654.28890)
  MoveL 9030 to (240.95, 148.22, 125.68) mm, rotated rx 180 ry 0 rz 180 deg; joints [-28.737, 15.299, 64.319, 71.807, 30.404, -69.14]
  MoveL 9031 to (240.95, 148.22, 125.68) mm, rotated rx 180 ry 0 rz 180 deg; joints [-28.737, 15.299, 64.319, 71.807, 30.404, -69.14]
  Call Extruder(654.48734)
  MoveL 9032 to (240.9, 148.6, 125.68) mm, rotated rx -180 ry 0 rz 180 deg; joints [-28.774, 15.326, 64.285, 71.822, 30.441, -69.15]
  MoveL 9033 to (240.9, 148.6, 125.68) mm, rotated rx -180 ry 0 rz 180 deg; joints [-28.774, 15.326, 64.285, 71.822, 30.441, -69.15]
  Call Extruder(654.68665)
  MoveL 9034 to (240.86, 148.99, 125.68) mm, rotated rx 180 ry 0 rz 180 deg; joints [-28.812, 15.353, 64.251, 71.837, 30.478, -69.16]
  MoveL 9035 to (240.86, 148.99, 125.68) mm, rotated rx 180 ry 0 rz 180 deg; joints [-28.812, 15.353, 64.251, 71.837, 30.478, -69.16]
  Call Extruder(654.84549)
  MoveL 9036 to (240.81, 149.3, 125.68) mm, rotated rx 180 ry 0 rz 180 deg; joints [-28.842, 15.373, 64.227, 71.85, 30.508, -69.169]
  MoveL 9037 to (240.81, 149.3, 125.68) mm, rotated rx 180 ry 0 rz 180 deg; joints [-28.842, 15.373, 64.227, 71.85, 30.508, -69.169]
  Call Extruder(655.00505)
  MoveL 9038 to (240.76, 149.6, 125.68) mm, rotated rx -180 ry 0 rz 180 deg; joints [-28.872, 15.392, 64.203, 71.864, 30.537, -69.178]
  MoveL 9039 to (240.76, 149.6, 125.68) mm, rotated rx -180 ry 0 rz 180 deg; joints [-28.872, 15.392, 64.203, 71.864, 30.537, -69.178]
  Call Extruder(655.16534)
  MoveL 9040 to (240.71, 149.91, 125.68) mm, rotated rx 180 ry 0 rz 180 deg; joints [-28.902, 15.411, 64.178, 71.877, 30.567, -69.187]
  MoveL 9041 to (240.71, 149.91, 125.68) mm, rotated rx 180 ry 0 rz 180 deg; joints [-28.902, 15.411, 64.178, 71.877, 30.567, -69.187]
  Call Extruder(655.32635)
  MoveL 9042 to (240.66, 150.21, 125.68) mm, rotated rx 180 ry 0 rz 180 deg; joints [-28.932, 15.431, 64.154, 71.89, 30.597, -69.196]
  MoveL 9043 to (240.66, 150.21, 125.68) mm, rotated rx 180 ry 0 rz 180 deg; joints [-28.932, 15.431, 64.154, 71.89, 30.597, -69.196]
  Call Extruder(655.48810)
  MoveL 9044 to (240.61, 150.52, 125.68) mm, rotated rx 180 ry 0 rz 180 deg; joints [-28.962, 15.45, 64.13, 71.903, 30.626, -69.205]
  MoveL 9045 to (240.61, 150.52, 125.68) mm, rotated rx 180 ry 0 rz 180 deg; joints [-28.962, 15.45, 64.13, 71.903, 30.626, -69.205]
  Call Extruder(655.65057)
  MoveL 9046 to (240.56, 150.83, 125.68) mm, rotated rx -180 ry 0 rz 180 deg; joints [-28.993, 15.47, 64.105, 71.916, 30.656, -69.213]
  MoveL 9047 to (240.56, 150.83, 125.68) mm, rotated rx -180 ry 0 rz 180 deg; joints [-28.993, 15.47, 64.105, 71.916, 30.656, -69.213]
  Call Extruder(655.78449)
  MoveL 9048 to (240.52, 151.08, 125.68) mm, rotated rx -180 ry 0 rz 180 deg; joints [-29.017, 15.484, 64.087, 71.927, 30.681, -69.222]
  MoveL 9049 to (240.52, 151.08, 125.68) mm, rotated rx -180 ry 0 rz 180 deg; joints [-29.017, 15.484, 64.087, 71.927, 30.681, -69.222]
  Call Extruder(655.91903)
  MoveL 9050 to (240.47, 151.32, 125.68) mm, rotated rx 180 ry 0 rz 180 deg; joints [-29.043, 15.498, 64.069, 71.939, 30.705, -69.23]
  MoveL 9051 to (240.47, 151.32, 125.68) mm, rotated rx 180 ry 0 rz 180 deg; joints [-29.043, 15.498, 64.069, 71.939, 30.705, -69.23]
  Call Extruder(656.05418)
  MoveL 9052 to (240.42, 151.57, 125.68) mm, rotated rx 180 ry 0 rz 180 deg; joints [-29.067, 15.513, 64.051, 71.95, 30.73, -69.238]
  MoveL 9053 to (240.42, 151.57, 125.68) mm, rotated rx 180 ry 0 rz 180 deg; joints [-29.067, 15.513, 64.051, 71.95, 30.73, -69.238]
  Call Extruder(656.18994)
  MoveL 9054 to (240.37, 151.82, 125.68) mm, rotated rx 180 ry 0 rz -180 deg; joints [-29.092, 15.527, 64.033, 71.962, 30.754, -69.246]
  MoveL 9055 to (240.37, 151.82, 125.68) mm, rotated rx 180 ry 0 rz -180 deg; joints [-29.092, 15.527, 64.033, 71.962, 30.754, -69.246]
  Call Extruder(656.32630)
  MoveL 9056 to (240.32, 152.07, 125.68) mm, rotated rx -180 ry 0 rz 180 deg; joints [-29.117, 15.541, 64.015, 71.973, 30.778, -69.254]
  MoveL 9057 to (240.32, 152.07, 125.68) mm, rotated rx -180 ry 0 rz 180 deg; joints [-29.117, 15.541, 64.015, 71.973, 30.778, -69.254]
  Call Extruder(656.46328)
  MoveL 9058 to (240.27, 152.32, 125.68) mm, rotated rx 180 ry 0 rz 180 deg; joints [-29.142, 15.556, 63.997, 71.985, 30.803, -69.262]
  MoveL 9059 to (240.27, 152.32, 125.68) mm, rotated rx 180 ry 0 rz 180 deg; joints [-29.142, 15.556, 63.997, 71.985, 30.803, -69.262]
  Call Extruder(656.60087)
  MoveL 9060 to (240.22, 152.57, 125.68) mm, rotated rx 180 ry 0 rz 180 deg; joints [-29.167, 15.57, 63.979, 71.996, 30.827, -69.27]
  MoveL 9061 to (240.22, 152.57, 125.68) mm, rotated rx 180 ry 0 rz 180 deg; joints [-29.167, 15.57, 63.979, 71.996, 30.827, -69.27]
  Call Extruder(656.71457)
  MoveL 9062 to (240.17, 152.77, 125.68) mm, rotated rx 180 ry 0 rz 180 deg; joints [-29.188, 15.582, 63.965, 72.006, 30.848, -69.277]
  MoveL 9063 to (240.17, 152.77, 125.68) mm, rotated rx 180 ry 0 rz 180 deg; joints [-29.188, 15.582, 63.965, 72.006, 30.848, -69.277]
  Call Extruder(656.82872)
  MoveL 9064 to (240.13, 152.98, 125.68) mm, rotated rx -180 ry 0 rz 180 deg; joints [-29.209, 15.593, 63.951, 72.015, 30.868, -69.284]
  MoveL 9065 to (240.13, 152.98, 125.68) mm, rotated rx -180 ry 0 rz 180 deg; joints [-29.209, 15.593, 63.951, 72.015, 30.868, -69.284]
  Call Extruder(656.94332)
  MoveL 9066 to (240.08, 153.18, 125.68) mm, rotated rx -180 ry 0 rz 180 deg; joints [-29.229, 15.604, 63.937, 72.025, 30.888, -69.291]
  MoveL 9067 to (240.08, 153.18, 125.68) mm, rotated rx -180 ry 0 rz 180 deg; joints [-29.229, 15.604, 63.937, 72.025, 30.888, -69.291]
  Call Extruder(657.05837)
  MoveL 9068 to (240.04, 153.39, 125.68) mm, rotated rx 180 ry 0 rz 180 deg; joints [-29.25, 15.615, 63.922, 72.035, 30.908, -69.297]
  MoveL 9069 to (240.04, 153.39, 125.68) mm, rotated rx 180 ry 0 rz 180 deg; joints [-29.25, 15.615, 63.922, 72.035, 30.908, -69.297]
  Call Extruder(657.18060)
  MoveL 9070 to (239.98, 153.6, 125.68) mm, rotated rx 180 ry 0 rz 180 deg; joints [-29.272, 15.625, 63.91, 72.046, 30.93, -69.305]
  MoveL 9071 to (239.98, 153.6, 125.68) mm, rotated rx 180 ry 0 rz 180 deg; joints [-29.272, 15.625, 63.91, 72.046, 30.93, -69.305]
  Call Extruder(657.31026)
  MoveL 9072 to (239.92, 153.82, 125.68) mm, rotated rx -180 ry 0 rz 180 deg; joints [-29.296, 15.635, 63.898, 72.058, 30.953, -69.315]
  MoveL 9073 to (239.92, 153.82, 125.68) mm, rotated rx -180 ry 0 rz 180 deg; joints [-29.296, 15.635, 63.898, 72.058, 30.953, -69.315]
  Call Extruder(657.44048)
  MoveL 9074 to (239.85, 154.05, 125.68) mm, rotated rx 180 ry 0 rz -180 deg; joints [-29.319, 15.644, 63.886, 72.07, 30.975, -69.324]
  MoveL 9075 to (239.85, 154.05, 125.68) mm, rotated rx 180 ry 0 rz -180 deg; joints [-29.319, 15.644, 63.886, 72.07, 30.975, -69.324]
  Call Extruder(657.57127)
  MoveL 9076 to (239.78, 154.27, 125.68) mm, rotated rx 180 ry 0 rz -180 deg; joints [-29.343, 15.653, 63.874, 72.083, 30.998, -69.334]
  MoveL 9077 to (239.78, 154.27, 125.68) mm, rotated rx 180 ry 0 rz -180 deg; joints [-29.343, 15.653, 63.874, 72.083, 30.998, -69.334]
  Call Extruder(657.70262)
  MoveL 9078 to (239.71, 154.5, 125.68) mm, rotated rx 180 ry 0 rz 180 deg; joints [-29.366, 15.663, 63.863, 72.095, 31.021, -69.343]
  MoveL 9079 to (239.71, 154.5, 125.68) mm, rotated rx 180 ry 0 rz 180 deg; joints [-29.366, 15.663, 63.863, 72.095, 31.021, -69.343]
  Call Extruder(657.81453)
  MoveL 9080 to (239.65, 154.68, 125.68) mm, rotated rx 180 ry 0 rz 180 deg; joints [-29.386, 15.67, 63.853, 72.106, 31.04, -69.351]
  MoveL 9081 to (239.65, 154.68, 125.68) mm, rotated rx 180 ry 0 rz 180 deg; joints [-29.386, 15.67, 63.853, 72.106, 31.04, -69.351]
  Call Extruder(657.92687)
  MoveL 9082 to (239.59, 154.87, 125.68) mm, rotated rx 180 ry 0 rz 180 deg; joints [-29.406, 15.677, 63.844, 72.116, 31.059, -69.36]
  MoveL 9083 to (239.59, 154.87, 125.68) mm, rotated rx 180 ry 0 rz 180 deg; joints [-29.406, 15.677, 63.844, 72.116, 31.059, -69.36]
  Call Extruder(658.03966)
  MoveL 9084 to (239.53, 155.06, 125.68) mm, rotated rx 180 ry 0 rz -180 deg; joints [-29.426, 15.684, 63.835, 72.127, 31.079, -69.368]
  MoveL 9085 to (239.53, 155.06, 125.68) mm, rotated rx 180 ry 0 rz -180 deg; joints [-29.426, 15.684, 63.835, 72.127, 31.079, -69.368]
  Call Extruder(658.15290)
  MoveL 9086 to (239.47, 155.25, 125.68) mm, rotated rx 180 ry 0 rz 180 deg; joints [-29.446, 15.692, 63.826, 72.138, 31.098, -69.376]
  MoveL 9087 to (239.47, 155.25, 125.68) mm, rotated rx 180 ry 0 rz 180 deg; joints [-29.446, 15.692, 63.826, 72.138, 31.098, -69.376]
  Call Extruder(658.26658)
  MoveL 9088 to (239.41, 155.44, 125.68) mm, rotated rx 180 ry 0 rz 180 deg; joints [-29.466, 15.699, 63.817, 72.148, 31.117, -69.384]
  MoveL 9089 to (239.41, 155.44, 125.68) mm, rotated rx 180 ry 0 rz 180 deg; joints [-29.466, 15.699, 63.817, 72.148, 31.117, -69.384]
  Call Extruder(658.44854)
  MoveL 9090 to (239.29, 155.73, 125.68) mm, rotated rx 180 ry 0 rz 180 deg; joints [-29.499, 15.706, 63.808, 72.168, 31.148, -69.4]
  MoveL 9091 to (239.29, 155.73, 125.68) mm, rotated rx 180 ry 0 rz 180 deg; joints [-29.499, 15.706, 63.808, 72.168, 31.148, -69.4]
  Call Extruder(658.63125)
  MoveL 9092 to (239.16, 156.02, 125.68) mm, rotated rx 180 ry 0 rz 180 deg; joints [-29.531, 15.713, 63.799, 72.187, 31.179, -69.415]
  MoveL 9093 to (239.16, 156.02, 125.68) mm, rotated rx 180 ry 0 rz 180 deg; joints [-29.531, 15.713, 63.799, 72.187, 31.179, -69.415]
  Call Extruder(658.80168)
  MoveL 9094 to (239.05, 156.29, 125.68) mm, rotated rx 180 ry 0 rz 180 deg; joints [-29.561, 15.72, 63.791, 72.204, 31.208, -69.43]
  MoveL 9095 to (239.05, 156.29, 125.68) mm, rotated rx 180 ry 0 rz 180 deg; joints [-29.561, 15.72, 63.791, 72.204, 31.208, -69.43]
  Call Extruder(658.95972)
  MoveL 9096 to (238.94, 156.54, 125.68) mm, rotated rx -180 ry 0 rz 180 deg; joints [-29.589, 15.725, 63.784, 72.221, 31.234, -69.443]
  MoveL 9097 to (238.94, 156.54, 125.68) mm, rotated rx -180 ry 0 rz 180 deg; joints [-29.589, 15.725, 63.784, 72.221, 31.234, -69.443]
  Call Extruder(659.11835)
  MoveL 9098 to (238.84, 156.79, 125.68) mm, rotated rx 180 ry 0 rz 180 deg; joints [-29.617, 15.731, 63.777, 72.238, 31.261, -69.457]
  MoveL 9099 to (238.84, 156.79, 125.68) mm, rotated rx 180 ry 0 rz 180 deg; joints [-29.617, 15.731, 63.777, 72.238, 31.261, -69.457]
  Call Extruder(659.32451)
  MoveL 9100 to (238.66, 157.09, 125.68) mm, rotated rx -180 ry 0 rz 180 deg; joints [-29.653, 15.73, 63.777, 72.262, 31.294, -69.478]
  MoveL 9101 to (238.66, 157.09, 125.68) mm, rotated rx -180 ry 0 rz 180 deg; joints [-29.653, 15.73, 63.777, 72.262, 31.294, -69.478]
  Call Extruder(659.53144)
  MoveL 9102 to (238.49, 157.4, 125.68) mm, rotated rx 180 ry 0 rz 180 deg; joints [-29.689, 15.73, 63.778, 72.287, 31.328, -69.499]
  MoveL 9103 to (238.49, 157.4, 125.68) mm, rotated rx 180 ry 0 rz 180 deg; joints [-29.689, 15.73, 63.778, 72.287, 31.328, -69.499]
  Call Extruder(659.73916)
  MoveL 9104 to (238.31, 157.7, 125.68) mm, rotated rx -180 ry 0 rz 180 deg; joints [-29.725, 15.73, 63.778, 72.311, 31.362, -69.52]
  MoveL 9105 to (238.31, 157.7, 125.68) mm, rotated rx -180 ry 0 rz 180 deg; joints [-29.725, 15.73, 63.778, 72.311, 31.362, -69.52]
  Call Extruder(659.94765)
  MoveL 9106 to (238.13, 158.01, 125.68) mm, rotated rx 180 ry 0 rz 180 deg; joints [-29.761, 15.729, 63.779, 72.336, 31.396, -69.54]
  MoveL 9107 to (238.13, 158.01, 125.68) mm, rotated rx 180 ry 0 rz 180 deg; joints [-29.761, 15.729, 63.779, 72.336, 31.396, -69.54]
  Call Extruder(660.12717)
  MoveL 9108 to (237.96, 158.25, 125.68) mm, rotated rx 180 ry 0 rz 180 deg; joints [-29.792, 15.724, 63.786, 72.359, 31.425, -69.561]
  MoveL 9109 to (237.96, 158.25, 125.68) mm, rotated rx 180 ry 0 rz 180 deg; joints [-29.792, 15.724, 63.786, 72.359, 31.425, -69.561]
  Call Extruder(660.46059)
  MoveL 9110 to (237.63, 158.7, 125.68) mm, rotated rx 180 ry 0 rz 180 deg; joints [-29.849, 15.713, 63.8, 72.401, 31.477, -69.599]
  MoveL 9111 to (237.63, 158.7, 125.68) mm, rotated rx 180 ry 0 rz 180 deg; joints [-29.849, 15.713, 63.8, 72.401, 31.477, -69.599]
  Call Extruder(660.79519)
  MoveL 9112 to (237.3, 159.15, 125.68) mm, rotated rx -180 ry 0 rz 180 deg; joints [-29.907, 15.702, 63.814, 72.444, 31.53, -69.637]
  Call Extruder(661.62314)
  MoveL 9113 to (236.39, 160.19, 125.68) mm, rotated rx 180 ry 0 rz 180 deg; joints [-30.046, 15.651, 63.877, 72.557, 31.657, -69.739]
  Call Extruder(662.45109)
  MoveL 9114 to (235.35, 161.1, 125.68) mm, rotated rx 180 ry 0 rz 180 deg; joints [-30.182, 15.57, 63.979, 72.678, 31.778, -69.852]
  Call Extruder(662.61839)
  MoveL 9115 to (235.13, 161.27, 125.68) mm, rotated rx 180 ry 0 rz -180 deg; joints [-30.208, 15.549, 64.005, 72.703, 31.801, -69.877]
  MoveL 9116 to (235.13, 161.27, 125.68) mm, rotated rx 180 ry 0 rz -180 deg; joints [-30.208, 15.549, 64.005, 72.703, 31.801, -69.877]
  Call Extruder(662.95182)
  MoveL 9117 to (234.68, 161.59, 125.68) mm, rotated rx 180 ry 0 rz 180 deg; joints [-30.261, 15.508, 64.058, 72.754, 31.847, -69.925]
  MoveL 9118 to (234.68, 161.59, 125.68) mm, rotated rx 180 ry 0 rz 180 deg; joints [-30.261, 15.508, 64.058, 72.754, 31.847, -69.925]
  Call Extruder(663.28405)
  MoveL 9119 to (234.23, 161.92, 125.68) mm, rotated rx 180 ry 0 rz -180 deg; joints [-30.314, 15.466, 64.11, 72.804, 31.894, -69.973]
  MoveL 9120 to (234.23, 161.92, 125.68) mm, rotated rx 180 ry 0 rz -180 deg; joints [-30.314, 15.466, 64.11, 72.804, 31.894, -69.973]
  Call Extruder(663.40172)
  MoveL 9121 to (234.05, 162.02, 125.68) mm, rotated rx 180 ry 0 rz 180 deg; joints [-30.331, 15.448, 64.132, 72.823, 31.909, -69.992]
  MoveL 9122 to (234.05, 162.02, 125.68) mm, rotated rx 180 ry 0 rz 180 deg; joints [-30.331, 15.448, 64.132, 72.823, 31.909, -69.992]
  Call Extruder(663.60945)
  MoveL 9123 to (233.75, 162.2, 125.68) mm, rotated rx 180 ry 0 rz -180 deg; joints [-30.363, 15.416, 64.172, 72.856, 31.937, -70.024]
  MoveL 9124 to (233.75, 162.2, 125.68) mm, rotated rx 180 ry 0 rz -180 deg; joints [-30.363, 15.416, 64.172, 72.856, 31.937, -70.024]
  Call Extruder(663.81640)
  MoveL 9125 to (233.45, 162.37, 125.68) mm, rotated rx 180 ry 0 rz 180 deg; joints [-30.394, 15.384, 64.212, 72.889, 31.964, -70.055]
  MoveL 9126 to (233.45, 162.37, 125.68) mm, rotated rx 180 ry 0 rz 180 deg; joints [-30.394, 15.384, 64.212, 72.889, 31.964, -70.055]
  Call Extruder(664.02257)
  MoveL 9127 to (233.14, 162.55, 125.68) mm, rotated rx 180 ry 0 rz 180 deg; joints [-30.426, 15.352, 64.252, 72.921, 31.991, -70.087]
  MoveL 9128 to (233.14, 162.55, 125.68) mm, rotated rx 180 ry 0 rz 180 deg; joints [-30.426, 15.352, 64.252, 72.921, 31.991, -70.087]
  Call Extruder(664.20424)
  MoveL 9129 to (232.87, 162.69, 125.68) mm, rotated rx 180 ry 0 rz 180 deg; joints [-30.453, 15.322, 64.291, 72.951, 32.014, -70.116]
  MoveL 9130 to (232.87, 162.69, 125.68) mm, rotated rx 180 ry 0 rz 180 deg; joints [-30.453, 15.322, 64.291, 72.951, 32.014, -70.116]
  Call Extruder(664.36221)
  MoveL 9131 to (232.62, 162.8, 125.68) mm, rotated rx -180 ry 0 rz 180 deg; joints [-30.476, 15.292, 64.328, 72.977, 32.033, -70.142]
  MoveL 9132 to (232.62, 162.8, 125.68) mm, rotated rx -180 ry 0 rz 180 deg; joints [-30.476, 15.292, 64.328, 72.977, 32.033, -70.142]
  Call Extruder(664.51957)
  MoveL 9133 to (232.37, 162.91, 125.68) mm, rotated rx 180 ry 0 rz 180 deg; joints [-30.498, 15.263, 64.365, 73.002, 32.052, -70.167]
  MoveL 9134 to (232.37, 162.91, 125.68) mm, rotated rx 180 ry 0 rz 180 deg; joints [-30.498, 15.263, 64.365, 73.002, 32.052, -70.167]
  Call Extruder(664.70231)
  MoveL 9135 to (232.08, 163.03, 125.68) mm, rotated rx -180 ry 0 rz 180 deg; joints [-30.524, 15.227, 64.409, 73.032, 32.074, -70.197]
  MoveL 9136 to (232.08, 163.03, 125.68) mm, rotated rx -180 ry 0 rz 180 deg; joints [-30.524, 15.227, 64.409, 73.032, 32.074, -70.197]
  Call Extruder(664.88429)
  MoveL 9137 to (231.78, 163.15, 125.68) mm, rotated rx 180 ry 0 rz -180 deg; joints [-30.551, 15.193, 64.452, 73.063, 32.097, -70.227]
  MoveL 9138 to (231.78, 163.15, 125.68) mm, rotated rx 180 ry 0 rz -180 deg; joints [-30.551, 15.193, 64.452, 73.063, 32.097, -70.227]
  Call Extruder(665.03163)
  MoveL 9139 to (231.54, 163.24, 125.68) mm, rotated rx 180 ry 0 rz 180 deg; joints [-30.571, 15.163, 64.489, 73.087, 32.114, -70.252]
  MoveL 9140 to (231.54, 163.24, 125.68) mm, rotated rx 180 ry 0 rz 180 deg; joints [-30.571, 15.163, 64.489, 73.087, 32.114, -70.252]
  Call Extruder(665.14485)
  MoveL 9141 to (231.35, 163.3, 125.68) mm, rotated rx 180 ry 0 rz 180 deg; joints [-30.587, 15.139, 64.519, 73.106, 32.127, -70.271]
  MoveL 9142 to (231.35, 163.3, 125.68) mm, rotated rx 180 ry 0 rz 180 deg; joints [-30.587, 15.139, 64.519, 73.106, 32.127, -70.271]
  Call Extruder(665.25763)
  MoveL 9143 to (231.17, 163.36, 125.68) mm, rotated rx -180 ry 0 rz 180 deg; joints [-30.602, 15.115, 64.549, 73.125, 32.139, -70.29]
  MoveL 9144 to (231.17, 163.36, 125.68) mm, rotated rx -180 ry 0 rz 180 deg; joints [-30.602, 15.115, 64.549, 73.125, 32.139, -70.29]
  Call Extruder(665.36996)
  MoveL 9145 to (230.98, 163.42, 125.68) mm, rotated rx 180 ry 0 rz -180 deg; joints [-30.618, 15.091, 64.579, 73.144, 32.152, -70.309]
  MoveL 9146 to (230.98, 163.42, 125.68) mm, rotated rx 180 ry 0 rz -180 deg; joints [-30.618, 15.091, 64.579, 73.144, 32.152, -70.309]
  Call Extruder(665.48185)
  MoveL 9147 to (230.79, 163.48, 125.68) mm, rotated rx 180 ry 0 rz 180 deg; joints [-30.633, 15.067, 64.609, 73.163, 32.165, -70.328]
  MoveL 9148 to (230.79, 163.48, 125.68) mm, rotated rx 180 ry 0 rz 180 deg; joints [-30.633, 15.067, 64.609, 73.163, 32.165, -70.328]
  Call Extruder(665.60326)
  MoveL 9149 to (230.58, 163.55, 125.68) mm, rotated rx -180 ry 0 rz 180 deg; joints [-30.65, 15.04, 64.642, 73.183, 32.179, -70.349]
  MoveL 9150 to (230.58, 163.55, 125.68) mm, rotated rx -180 ry 0 rz 180 deg; joints [-30.65, 15.04, 64.642, 73.183, 32.179, -70.349]
  Call Extruder(665.73407)
  MoveL 9151 to (230.36, 163.62, 125.68) mm, rotated rx -180 ry 0 rz 180 deg; joints [-30.668, 15.012, 64.678, 73.205, 32.194, -70.371]
  MoveL 9152 to (230.36, 163.62, 125.68) mm, rotated rx -180 ry 0 rz 180 deg; joints [-30.668, 15.012, 64.678, 73.205, 32.194, -70.371]
  Call Extruder(665.86432)
  MoveL 9153 to (230.14, 163.68, 125.68) mm, rotated rx -180 ry 0 rz 180 deg; joints [-30.685, 14.983, 64.714, 73.227, 32.208, -70.393]
  MoveL 9154 to (230.14, 163.68, 125.68) mm, rotated rx -180 ry 0 rz 180 deg; joints [-30.685, 14.983, 64.714, 73.227, 32.208, -70.393]
  Call Extruder(665.99400)
  MoveL 9155 to (229.91, 163.75, 125.68) mm, rotated rx 180 ry 0 rz 180 deg; joints [-30.703, 14.954, 64.75, 73.249, 32.223, -70.416]
  MoveL 9156 to (229.91, 163.75, 125.68) mm, rotated rx 180 ry 0 rz 180 deg; joints [-30.703, 14.954, 64.75, 73.249, 32.223, -70.416]
  Call Extruder(666.12312)
  MoveL 9157 to (229.69, 163.82, 125.68) mm, rotated rx 180 ry 0 rz 180 deg; joints [-30.721, 14.925, 64.787, 73.271, 32.238, -70.438]
  MoveL 9158 to (229.69, 163.82, 125.68) mm, rotated rx 180 ry 0 rz 180 deg; joints [-30.721, 14.925, 64.787, 73.271, 32.238, -70.438]
  Call Extruder(666.23819)
  MoveL 9159 to (229.48, 163.86, 125.68) mm, rotated rx -180 ry 0 rz 180 deg; joints [-30.736, 14.897, 64.821, 73.291, 32.25, -70.458]
  MoveL 9160 to (229.48, 163.86, 125.68) mm, rotated rx -180 ry 0 rz 180 deg; joints [-30.736, 14.897, 64.821, 73.291, 32.25, -70.458]
  Call Extruder(666.35282)
  MoveL 9161 to (229.28, 163.91, 125.68) mm, rotated rx 180 ry 0 rz 180 deg; joints [-30.751, 14.869, 64.856, 73.311, 32.262, -70.478]
  MoveL 9162 to (229.28, 163.91, 125.68) mm, rotated rx 180 ry 0 rz 180 deg; joints [-30.751, 14.869, 64.856, 73.311, 32.262, -70.478]
  Call Extruder(666.46699)
  MoveL 9163 to (229.08, 163.95, 125.68) mm, rotated rx -180 ry 0 rz 180 deg; joints [-30.766, 14.841, 64.891, 73.33, 32.274, -70.498]
  MoveL 9164 to (229.08, 163.95, 125.68) mm, rotated rx -180 ry 0 rz 180 deg; joints [-30.766, 14.841, 64.891, 73.33, 32.274, -70.498]
  Call Extruder(666.58070)
  MoveL 9165 to (228.87, 164, 125.68) mm, rotated rx 180 ry 0 rz 180 deg; joints [-30.781, 14.813, 64.926, 73.35, 32.286, -70.519]
  MoveL 9166 to (228.87, 164, 125.68) mm, rotated rx 180 ry 0 rz 180 deg; joints [-30.781, 14.813, 64.926, 73.35, 32.286, -70.519]
  Call Extruder(666.70613)
  MoveL 9167 to (228.65, 164.04, 125.68) mm, rotated rx 180 ry 0 rz 180 deg; joints [-30.797, 14.782, 64.964, 73.372, 32.299, -70.541]
  MoveL 9168 to (228.65, 164.04, 125.68) mm, rotated rx 180 ry 0 rz 180 deg; joints [-30.797, 14.782, 64.964, 73.372, 32.299, -70.541]
  Call Extruder(666.84310)
  MoveL 9169 to (228.4, 164.09, 125.68) mm, rotated rx 180 ry 0 rz 180 deg; joints [-30.815, 14.748, 65.007, 73.396, 32.314, -70.565]
  MoveL 9170 to (228.4, 164.09, 125.68) mm, rotated rx 180 ry 0 rz 180 deg; joints [-30.815, 14.748, 65.007, 73.396, 32.314, -70.565]
  Call Extruder(666.97947)
  MoveL 9171 to (228.15, 164.14, 125.68) mm, rotated rx 180 ry 0 rz 180 deg; joints [-30.832, 14.713, 65.05, 73.419, 32.328, -70.589]
  MoveL 9172 to (228.15, 164.14, 125.68) mm, rotated rx 180 ry 0 rz 180 deg; joints [-30.832, 14.713, 65.05, 73.419, 32.328, -70.589]
  Call Extruder(667.11523)
  MoveL 9173 to (227.9, 164.19, 125.68) mm, rotated rx 180 ry 0 rz 180 deg; joints [-30.85, 14.679, 65.092, 73.443, 32.342, -70.614]
  MoveL 9174 to (227.9, 164.19, 125.68) mm, rotated rx 180 ry 0 rz 180 deg; joints [-30.85, 14.679, 65.092, 73.443, 32.342, -70.614]
  Call Extruder(667.25038)
  MoveL 9175 to (227.65, 164.24, 125.68) mm, rotated rx 180 ry 0 rz 180 deg; joints [-30.868, 14.644, 65.135, 73.466, 32.357, -70.638]
  MoveL 9176 to (227.65, 164.24, 125.68) mm, rotated rx 180 ry 0 rz 180 deg; joints [-30.868, 14.644, 65.135, 73.466, 32.357, -70.638]
  Call Extruder(667.38491)
  MoveL 9177 to (227.4, 164.29, 125.68) mm, rotated rx 180 ry 0 rz 180 deg; joints [-30.886, 14.61, 65.178, 73.49, 32.371, -70.662]
  MoveL 9178 to (227.4, 164.29, 125.68) mm, rotated rx 180 ry 0 rz 180 deg; joints [-30.886, 14.61, 65.178, 73.49, 32.371, -70.662]
  Call Extruder(667.51884)
  MoveL 9179 to (227.15, 164.34, 125.68) mm, rotated rx 180 ry 0 rz -180 deg; joints [-30.903, 14.576, 65.22, 73.513, 32.385, -70.686]
  MoveL 9180 to (227.15, 164.34, 125.68) mm, rotated rx 180 ry 0 rz -180 deg; joints [-30.903, 14.576, 65.22, 73.513, 32.385, -70.686]
  Call Extruder(667.66670)
  MoveL 9181 to (226.87, 164.39, 125.68) mm, rotated rx -180 ry 0 rz -180 deg; joints [-30.923, 14.537, 65.268, 73.539, 32.401, -70.712]
  MoveL 9182 to (226.87, 164.39, 125.68) mm, rotated rx -180 ry 0 rz -180 deg; joints [-30.923, 14.537, 65.268, 73.539, 32.401, -70.712]
  Call Extruder(667.82844)
  MoveL 9183 to (226.57, 164.44, 125.68) mm, rotated rx 180 ry 0 rz 180 deg; joints [-30.943, 14.494, 65.322, 73.568, 32.418, -70.742]
  MoveL 9184 to (226.57, 164.44, 125.68) mm, rotated rx 180 ry 0 rz 180 deg; joints [-30.943, 14.494, 65.322, 73.568, 32.418, -70.742]
  Call Extruder(667.98945)
  MoveL 9185 to (226.26, 164.49, 125.68) mm, rotated rx -180 ry 0 rz -180 deg; joints [-30.964, 14.451, 65.375, 73.596, 32.434, -70.771]
  MoveL 9186 to (226.26, 164.49, 125.68) mm, rotated rx -180 ry 0 rz -180 deg; joints [-30.964, 14.451, 65.375, 73.596, 32.434, -70.771]
  Call Extruder(668.14974)
  MoveL 9187 to (225.95, 164.54, 125.68) mm, rotated rx 180 ry 0 rz 180 deg; joints [-30.985, 14.408, 65.428, 73.624, 32.451, -70.8]
  MoveL 9188 to (225.95, 164.54, 125.68) mm, rotated rx 180 ry 0 rz 180 deg; joints [-30.985, 14.408, 65.428, 73.624, 32.451, -70.8]
  Call Extruder(668.30929)
  MoveL 9189 to (225.65, 164.58, 125.68) mm, rotated rx 180 ry 0 rz 180 deg; joints [-31.006, 14.365, 65.482, 73.652, 32.468, -70.829]
  MoveL 9190 to (225.65, 164.58, 125.68) mm, rotated rx 180 ry 0 rz 180 deg; joints [-31.006, 14.365, 65.482, 73.652, 32.468, -70.829]
  Call Extruder(668.46812)
  MoveL 9191 to (225.34, 164.63, 125.68) mm, rotated rx 180 ry 0 rz -180 deg; joints [-31.027, 14.322, 65.535, 73.68, 32.485, -70.858]
  MoveL 9192 to (225.34, 164.63, 125.68) mm, rotated rx 180 ry 0 rz -180 deg; joints [-31.027, 14.322, 65.535, 73.68, 32.485, -70.858]
  Call Extruder(668.64679)
  MoveL 9193 to (225, 164.68, 125.68) mm, rotated rx 180 ry 0 rz 180 deg; joints [-31.049, 14.272, 65.596, 73.712, 32.503, -70.89]
  MoveL 9194 to (225, 164.68, 125.68) mm, rotated rx 180 ry 0 rz 180 deg; joints [-31.049, 14.272, 65.596, 73.712, 32.503, -70.89]
  Call Extruder(668.84523)
  MoveL 9195 to (224.61, 164.73, 125.68) mm, rotated rx 180 ry 0 rz -180 deg; joints [-31.074, 14.217, 65.665, 73.747, 32.523, -70.927]
  MoveL 9196 to (224.61, 164.73, 125.68) mm, rotated rx 180 ry 0 rz -180 deg; joints [-31.074, 14.217, 65.665, 73.747, 32.523, -70.927]
  Call Extruder(669.04281)
  MoveL 9197 to (224.22, 164.77, 125.68) mm, rotated rx -180 ry 0 rz 180 deg; joints [-31.1, 14.161, 65.734, 73.781, 32.543, -70.963]
  MoveL 9198 to (224.22, 164.77, 125.68) mm, rotated rx -180 ry 0 rz 180 deg; joints [-31.1, 14.161, 65.734, 73.781, 32.543, -70.963]
  Call Extruder(669.23952)
  MoveL 9199 to (223.83, 164.82, 125.68) mm, rotated rx 180 ry 0 rz 180 deg; joints [-31.125, 14.105, 65.802, 73.816, 32.563, -70.999]
  MoveL 9200 to (223.83, 164.82, 125.68) mm, rotated rx 180 ry 0 rz 180 deg; joints [-31.125, 14.105, 65.802, 73.816, 32.563, -70.999]
  Call Extruder(669.43535)
  MoveL 9201 to (223.45, 164.86, 125.68) mm, rotated rx 180 ry 0 rz 180 deg; joints [-31.15, 14.049, 65.871, 73.851, 32.583, -71.034]
  MoveL 9202 to (223.45, 164.86, 125.68) mm, rotated rx 180 ry 0 rz 180 deg; joints [-31.15, 14.049, 65.871, 73.851, 32.583, -71.034]
  Call Extruder(669.73071)
  MoveL 9203 to (222.86, 164.91, 125.68) mm, rotated rx 180 ry 0 rz 180 deg; joints [-31.186, 13.963, 65.977, 73.903, 32.612, -71.088]
  MoveL 9204 to (222.86, 164.91, 125.68) mm, rotated rx 180 ry 0 rz 180 deg; joints [-31.186, 13.963, 65.977, 73.903, 32.612, -71.088]
  Call Extruder(670.02474)
  MoveL 9205 to (222.27, 164.95, 125.68) mm, rotated rx -180 ry 0 rz 180 deg; joints [-31.222, 13.876, 66.084, 73.954, 32.641, -71.142]
  MoveL 9206 to (222.27, 164.95, 125.68) mm, rotated rx -180 ry 0 rz 180 deg; joints [-31.222, 13.876, 66.084, 73.954, 32.641, -71.142]
  Call Extruder(670.31744)
  MoveL 9207 to (221.68, 165, 125.68) mm, rotated rx 180 ry 0 rz 180 deg; joints [-31.258, 13.79, 66.19, 74.005, 32.67, -71.195]
  MoveL 9208 to (221.68, 165, 125.68) mm, rotated rx 180 ry 0 rz 180 deg; joints [-31.258, 13.79, 66.19, 74.005, 32.67, -71.195]
  Call Extruder(670.89088)
  MoveL 9209 to (220.52, 165.05, 125.68) mm, rotated rx -180 ry 0 rz 180 deg; joints [-31.326, 13.615, 66.404, 74.104, 32.723, -71.299]
  MoveL 9210 to (220.52, 165.05, 125.68) mm, rotated rx -180 ry 0 rz 180 deg; joints [-31.326, 13.615, 66.404, 74.104, 32.723, -71.299]
  Call Extruder(671.60489)
  MoveL 9211 to (219.06, 165.09, 125.68) mm, rotated rx -180 ry 0 rz 180 deg; joints [-31.409, 13.396, 66.671, 74.227, 32.789, -71.427]
  Call Extruder(788.45163)
  MoveL 9212 to (-19.06, 165.09, 125.68) mm, rotated rx 180 ry 0 rz -180 deg; joints [-51.475, -15.174, 94.824, 81.859, 52.214, -76.859]
  Call Extruder(788.88023)
  MoveL 9213 to (-19.94, 165.07, 125.68) mm, rotated rx 180 ry 0 rz 180 deg; joints [-51.582, -15.256, 94.885, 81.874, 52.321, -76.852]
  MoveL 9214 to (-19.94, 165.07, 125.68) mm, rotated rx 180 ry 0 rz 180 deg; joints [-51.582, -15.256, 94.885, 81.874, 52.321, -76.852]
  Call Extruder(789.45369)
  MoveL 9215 to (-21.1, 165.03, 125.68) mm, rotated rx -180 ry 0 rz 180 deg; joints [-51.722, -15.366, 94.967, 81.894, 52.461, -76.842]
  MoveL 9216 to (-21.1, 165.03, 125.68) mm, rotated rx -180 ry 0 rz 180 deg; joints [-51.722, -15.366, 94.967, 81.894, 52.461, -76.842]
  Call Extruder(789.88798)
  MoveL 9217 to (-21.97, 164.98, 125.68) mm, rotated rx 180 ry 0 rz 180 deg; joints [-51.827, -15.45, 95.03, 81.907, 52.566, -76.834]
  MoveL 9218 to (-21.97, 164.98, 125.68) mm, rotated rx 180 ry 0 rz 180 deg; joints [-51.827, -15.45, 95.03, 81.907, 52.566, -76.834]
  Call Extruder(790.18201)
  MoveL 9219 to (-22.56, 164.93, 125.68) mm, rotated rx 180 ry 0 rz 180 deg; joints [-51.897, -15.509, 95.074, 81.916, 52.636, -76.827]
  MoveL 9220 to (-22.56, 164.93, 125.68) mm, rotated rx 180 ry 0 rz 180 deg; joints [-51.897, -15.509, 95.074, 81.916, 52.636, -76.827]
  Call Extruder(790.47737)
  MoveL 9221 to (-23.15, 164.89, 125.68) mm, rotated rx 180 ry 0 rz 180 deg; joints [-51.966, -15.567, 95.117, 81.925, 52.706, -76.821]
  MoveL 9222 to (-23.15, 164.89, 125.68) mm, rotated rx 180 ry 0 rz 180 deg; joints [-51.966, -15.567, 95.117, 81.925, 52.706, -76.821]
  Call Extruder(790.72359)
  MoveL 9223 to (-23.64, 164.84, 125.68) mm, rotated rx -180 ry 0 rz 180 deg; joints [-52.023, -15.616, 95.154, 81.931, 52.763, -76.815]
  MoveL 9224 to (-23.64, 164.84, 125.68) mm, rotated rx -180 ry 0 rz 180 deg; joints [-52.023, -15.616, 95.154, 81.931, 52.763, -76.815]
  Call Extruder(790.92030)
  MoveL 9225 to (-24.03, 164.79, 125.68) mm, rotated rx 180 ry 0 rz 180 deg; joints [-52.067, -15.656, 95.183, 81.936, 52.807, -76.81]
  MoveL 9226 to (-24.03, 164.79, 125.68) mm, rotated rx 180 ry 0 rz 180 deg; joints [-52.067, -15.656, 95.183, 81.936, 52.807, -76.81]
  Call Extruder(791.11787)
  MoveL 9227 to (-24.42, 164.75, 125.68) mm, rotated rx 180 ry 0 rz -180 deg; joints [-52.112, -15.696, 95.213, 81.941, 52.852, -76.805]
  MoveL 9228 to (-24.42, 164.75, 125.68) mm, rotated rx 180 ry 0 rz -180 deg; joints [-52.112, -15.696, 95.213, 81.941, 52.852, -76.805]
  Call Extruder(791.31631)
  MoveL 9229 to (-24.8, 164.7, 125.68) mm, rotated rx -180 ry 0 rz -180 deg; joints [-52.156, -15.736, 95.243, 81.946, 52.897, -76.8]
  MoveL 9230 to (-24.8, 164.7, 125.68) mm, rotated rx -180 ry 0 rz -180 deg; joints [-52.156, -15.736, 95.243, 81.946, 52.897, -76.8]
  Call Extruder(791.51562)
  MoveL 9231 to (-25.19, 164.66, 125.68) mm, rotated rx -180 ry 0 rz -180 deg; joints [-52.2, -15.776, 95.272, 81.951, 52.942, -76.794]
  MoveL 9232 to (-25.19, 164.66, 125.68) mm, rotated rx -180 ry 0 rz -180 deg; joints [-52.2, -15.776, 95.272, 81.951, 52.942, -76.794]
  Call Extruder(791.67445)
  MoveL 9233 to (-25.5, 164.61, 125.68) mm, rotated rx -180 ry 0 rz 180 deg; joints [-52.235, -15.809, 95.296, 81.955, 52.976, -76.79]
  MoveL 9234 to (-25.5, 164.61, 125.68) mm, rotated rx -180 ry 0 rz 180 deg; joints [-52.235, -15.809, 95.296, 81.955, 52.976, -76.79]
  Call Extruder(791.83401)
  MoveL 9235 to (-25.8, 164.56, 125.68) mm, rotated rx 180 ry 0 rz 180 deg; joints [-52.269, -15.842, 95.321, 81.958, 53.01, -76.785]
  MoveL 9236 to (-25.8, 164.56, 125.68) mm, rotated rx 180 ry 0 rz 180 deg; joints [-52.269, -15.842, 95.321, 81.958, 53.01, -76.785]
  Call Extruder(791.99430)
  MoveL 9237 to (-26.11, 164.51, 125.68) mm, rotated rx -180 ry 0 rz 180 deg; joints [-52.303, -15.874, 95.345, 81.961, 53.045, -76.78]
  MoveL 9238 to (-26.11, 164.51, 125.68) mm, rotated rx -180 ry 0 rz 180 deg; joints [-52.303, -15.874, 95.345, 81.961, 53.045, -76.78]
  Call Extruder(792.15531)
  MoveL 9239 to (-26.41, 164.46, 125.68) mm, rotated rx 180 ry 0 rz 180 deg; joints [-52.337, -15.907, 95.369, 81.965, 53.079, -76.775]
  MoveL 9240 to (-26.41, 164.46, 125.68) mm, rotated rx 180 ry 0 rz 180 deg; joints [-52.337, -15.907, 95.369, 81.965, 53.079, -76.775]
  Call Extruder(792.31706)
  MoveL 9241 to (-26.72, 164.41, 125.68) mm, rotated rx 180 ry 0 rz -180 deg; joints [-52.371, -15.94, 95.393, 81.968, 53.113, -76.771]
  MoveL 9242 to (-26.72, 164.41, 125.68) mm, rotated rx 180 ry 0 rz -180 deg; joints [-52.371, -15.94, 95.393, 81.968, 53.113, -76.771]
  Call Extruder(792.47953)
  MoveL 9243 to (-27.02, 164.37, 125.68) mm, rotated rx 180 ry 0 rz 180 deg; joints [-52.405, -15.973, 95.417, 81.972, 53.148, -76.766]
  MoveL 9244 to (-27.02, 164.37, 125.68) mm, rotated rx 180 ry 0 rz 180 deg; joints [-52.405, -15.973, 95.417, 81.972, 53.148, -76.766]
  Call Extruder(792.61345)
  MoveL 9245 to (-27.27, 164.32, 125.68) mm, rotated rx 180 ry 0 rz 180 deg; joints [-52.432, -16.001, 95.438, 81.974, 53.175, -76.761]
  MoveL 9246 to (-27.27, 164.32, 125.68) mm, rotated rx 180 ry 0 rz 180 deg; joints [-52.432, -16.001, 95.438, 81.974, 53.175, -76.761]
  Call Extruder(792.74799)
  MoveL 9247 to (-27.52, 164.27, 125.68) mm, rotated rx 180 ry 0 rz 180 deg; joints [-52.459, -16.028, 95.458, 81.976, 53.202, -76.757]
  MoveL 9248 to (-27.52, 164.27, 125.68) mm, rotated rx 180 ry 0 rz 180 deg; joints [-52.459, -16.028, 95.458, 81.976, 53.202, -76.757]
  Call Extruder(792.88314)
  MoveL 9249 to (-27.77, 164.22, 125.68) mm, rotated rx 180 ry 0 rz 180 deg; joints [-52.486, -16.056, 95.479, 81.978, 53.23, -76.752]
  MoveL 9250 to (-27.77, 164.22, 125.68) mm, rotated rx 180 ry 0 rz 180 deg; joints [-52.486, -16.056, 95.479, 81.978, 53.23, -76.752]
  Call Extruder(793.01889)
  MoveL 9251 to (-28.02, 164.17, 125.68) mm, rotated rx 180 ry 0 rz -180 deg; joints [-52.513, -16.084, 95.499, 81.981, 53.257, -76.748]
  MoveL 9252 to (-28.02, 164.17, 125.68) mm, rotated rx 180 ry 0 rz -180 deg; joints [-52.513, -16.084, 95.499, 81.981, 53.257, -76.748]
  Call Extruder(793.15526)
  MoveL 9253 to (-28.27, 164.12, 125.68) mm, rotated rx 180 ry 0 rz 180 deg; joints [-52.54, -16.112, 95.52, 81.983, 53.284, -76.744]
  MoveL 9254 to (-28.27, 164.12, 125.68) mm, rotated rx 180 ry 0 rz 180 deg; joints [-52.54, -16.112, 95.52, 81.983, 53.284, -76.744]
  Call Extruder(793.24012)
  MoveL 9255 to (-28.42, 164.09, 125.68) mm, rotated rx -180 ry 0 rz -180 deg; joints [-52.556, -16.129, 95.532, 81.984, 53.301, -76.741]
  Set speed (130.0 mm/s)
  MoveL 9256 to (-31.76, 163.31, 125.68) mm, rotated rx 180 ry 0 rz 180 deg; joints [-52.91, -16.512, 95.813, 82.01, 53.659, -76.674]
  MoveL 9257 to (-31.76, 163.31, 135.08) mm, rotated rx 180 ry 0 rz -180 deg; joints [-52.91, -17.083, 97.633, 82.924, 53.495, -78.214]
  Call Extruder(791.24012)
  Set speed (40.0 mm/s)
  MoveL 9258 to (-31.76, 163.31, 135.08) mm, rotated rx 180 ry 0 rz -180 deg; joints [-52.91, -17.083, 97.633, 82.924, 53.495, -78.214]
  Call Extruder(0.00000)
  Set speed (130.0 mm/s)
  MoveL 9259 to (-39.41, 155.44, 135.08) mm, rotated rx 180 ry 0 rz 180 deg; joints [-53.137, -18.67, 98.757, 82.645, 53.776, -77.678]
  Call Extruder(2.00000)
  Set speed (40.0 mm/s)
  MoveL 9260 to (-39.41, 155.44, 135.08) mm, rotated rx 180 ry 0 rz 180 deg; joints [-53.137, -18.67, 98.757, 82.645, 53.776, -77.678]
  Set speed (30.0 mm/s)
  MoveL 9261 to (-39.41, 155.44, 135.08) mm, rotated rx 180 ry 0 rz 180 deg; joints [-53.137, -18.67, 98.757, 82.645, 53.776, -77.678]
  Call Extruder(2.05684)
  MoveL 9262 to (-39.44, 155.34, 135.08) mm, rotated rx 180 ry 0 rz 180 deg; joints [-53.131, -18.683, 98.766, 82.64, 53.771, -77.672]
  MoveL 9263 to (-39.44, 155.34, 135.08) mm, rotated rx 180 ry 0 rz 180 deg; joints [-53.131, -18.683, 98.766, 82.64, 53.771, -77.672]
  Call Extruder(2.17007)
  MoveL 9264 to (-39.5, 155.15, 135.08) mm, rotated rx -180 ry 0 rz 180 deg; joints [-53.121, -18.711, 98.785, 82.631, 53.761, -77.66]
  MoveL 9265 to (-39.5, 155.15, 135.08) mm, rotated rx -180 ry 0 rz 180 deg; joints [-53.121, -18.711, 98.785, 82.631, 53.761, -77.66]
  Call Extruder(2.28286)
  MoveL 9266 to (-39.56, 154.97, 135.08) mm, rotated rx 180 ry 0 rz 180 deg; joints [-53.11, -18.738, 98.804, 82.622, 53.752, -77.648]
  MoveL 9267 to (-39.56, 154.97, 135.08) mm, rotated rx 180 ry 0 rz 180 deg; joints [-53.11, -18.738, 98.804, 82.622, 53.752, -77.648]
  Call Extruder(2.39521)
  MoveL 9268 to (-39.62, 154.78, 135.08) mm, rotated rx 180 ry 0 rz 180 deg; joints [-53.099, -18.765, 98.823, 82.614, 53.742, -77.636]
  MoveL 9269 to (-39.62, 154.78, 135.08) mm, rotated rx 180 ry 0 rz 180 deg; joints [-53.099, -18.765, 98.823, 82.614, 53.742, -77.636]
  Call Extruder(2.50711)
  MoveL 9270 to (-39.68, 154.59, 135.08) mm, rotated rx 180 ry 0 rz 180 deg; joints [-53.088, -18.792, 98.842, 82.605, 53.733, -77.624]
  MoveL 9271 to (-39.68, 154.59, 135.08) mm, rotated rx 180 ry 0 rz 180 deg; joints [-53.088, -18.792, 98.842, 82.605, 53.733, -77.624]
  Call Extruder(2.62851)
  MoveL 9272 to (-39.75, 154.38, 135.08) mm, rotated rx -180 ry 0 rz 180 deg; joints [-53.076, -18.822, 98.862, 82.595, 53.722, -77.611]
  MoveL 9273 to (-39.75, 154.38, 135.08) mm, rotated rx -180 ry 0 rz 180 deg; joints [-53.076, -18.822, 98.862, 82.595, 53.722, -77.611]
  Call Extruder(2.75930)
  MoveL 9274 to (-39.82, 154.16, 135.08) mm, rotated rx 180 ry 0 rz 180 deg; joints [-53.063, -18.854, 98.884, 82.584, 53.71, -77.597]
  MoveL 9275 to (-39.82, 154.16, 135.08) mm, rotated rx 180 ry 0 rz 180 deg; joints [-53.063, -18.854, 98.884, 82.584, 53.71, -77.597]
  Call Extruder(2.88953)
  MoveL 9276 to (-39.88, 153.94, 135.08) mm, rotated rx 180 ry 0 rz 180 deg; joints [-53.049, -18.886, 98.906, 82.573, 53.698, -77.583]
  MoveL 9277 to (-39.88, 153.94, 135.08) mm, rotated rx 180 ry 0 rz 180 deg; joints [-53.049, -18.886, 98.906, 82.573, 53.698, -77.583]
  Call Extruder(3.01920)
  MoveL 9278 to (-39.95, 153.71, 135.08) mm, rotated rx -180 ry 0 rz 180 deg; joints [-53.036, -18.918, 98.929, 82.563, 53.687, -77.569]
  MoveL 9279 to (-39.95, 153.71, 135.08) mm, rotated rx -180 ry 0 rz 180 deg; joints [-53.036, -18.918, 98.929, 82.563, 53.687, -77.569]
  Call Extruder(3.14830)
  MoveL 9280 to (-40.02, 153.49, 135.08) mm, rotated rx 180 ry 0 rz 180 deg; joints [-53.022, -18.949, 98.951, 82.552, 53.674, -77.554]
  MoveL 9281 to (-40.02, 153.49, 135.08) mm, rotated rx 180 ry 0 rz 180 deg; joints [-53.022, -18.949, 98.951, 82.552, 53.674, -77.554]
  Call Extruder(3.26338)
  MoveL 9282 to (-40.06, 153.28, 135.08) mm, rotated rx 180 ry 0 rz 180 deg; joints [-53.007, -18.977, 98.97, 82.542, 53.661, -77.542]
  MoveL 9283 to (-40.06, 153.28, 135.08) mm, rotated rx 180 ry 0 rz 180 deg; joints [-53.007, -18.977, 98.97, 82.542, 53.661, -77.542]
  Call Extruder(3.37800)
  MoveL 9284 to (-40.11, 153.08, 135.08) mm, rotated rx 180 ry 0 rz 180 deg; joints [-52.993, -19.005, 98.989, 82.531, 53.648, -77.529]
  MoveL 9285 to (-40.11, 153.08, 135.08) mm, rotated rx 180 ry 0 rz 180 deg; joints [-52.993, -19.005, 98.989, 82.531, 53.648, -77.529]
  Call Extruder(3.49217)
  MoveL 9286 to (-40.15, 152.88, 135.08) mm, rotated rx 180 ry 0 rz 180 deg; joints [-52.978, -19.032, 99.008, 82.521, 53.635, -77.516]
  MoveL 9287 to (-40.15, 152.88, 135.08) mm, rotated rx 180 ry 0 rz 180 deg; joints [-52.978, -19.032, 99.008, 82.521, 53.635, -77.516]
  Call Extruder(3.60589)
  MoveL 9288 to (-40.2, 152.67, 135.08) mm, rotated rx -180 ry 0 rz 180 deg; joints [-52.963, -19.06, 99.027, 82.511, 53.621, -77.503]
  MoveL 9289 to (-40.2, 152.67, 135.08) mm, rotated rx -180 ry 0 rz 180 deg; joints [-52.963, -19.06, 99.027, 82.511, 53.621, -77.503]
  Call Extruder(3.70891)
  MoveL 9290 to (-40.23, 152.48, 135.08) mm, rotated rx -180 ry 0 rz 180 deg; joints [-52.949, -19.085, 99.044, 82.502, 53.609, -77.491]
  MoveL 9291 to (-40.23, 152.48, 135.08) mm, rotated rx -180 ry 0 rz 180 deg; joints [-52.949, -19.085, 99.044, 82.502, 53.609, -77.491]
  Call Extruder(3.80140)
  MoveL 9292 to (-40.27, 152.32, 135.08) mm, rotated rx 180 ry 0 rz 180 deg; joints [-52.937, -19.107, 99.059, 82.493, 53.598, -77.481]
  Set speed (130.0 mm/s)
  MoveL 9293 to (-40.27, 152.32, 135.08) mm, rotated rx 180 ry 0 rz 180 deg; joints [-52.937, -19.107, 99.059, 82.493, 53.598, -77.481]
  Set speed (30.0 mm/s)
  MoveL 9294 to (-40.27, 152.32, 135.08) mm, rotated rx 180 ry 0 rz 180 deg; joints [-52.937, -19.107, 99.059, 82.493, 53.598, -77.481]
  Call Extruder(3.93780)
  MoveL 9295 to (-40.32, 152.07, 135.08) mm, rotated rx -180 ry 0 rz 180 deg; joints [-52.918, -19.14, 99.082, 82.48, 53.581, -77.465]
  MoveL 9296 to (-40.32, 152.07, 135.08) mm, rotated rx -180 ry 0 rz 180 deg; joints [-52.918, -19.14, 99.082, 82.48, 53.581, -77.465]
  Call Extruder(4.07360)
  MoveL 9297 to (-40.37, 151.82, 135.08) mm, rotated rx 180 ry 0 rz 180 deg; joints [-52.899, -19.173, 99.105, 82.468, 53.564, -77.449]
  MoveL 9298 to (-40.37, 151.82, 135.08) mm, rotated rx 180 ry 0 rz 180 deg; joints [-52.899, -19.173, 99.105, 82.468, 53.564, -77.449]
  Call Extruder(4.20879)
  MoveL 9299 to (-40.42, 151.57, 135.08) mm, rotated rx -180 ry 0 rz 180 deg; joints [-52.881, -19.207, 99.128, 82.455, 53.547, -77.433]
  MoveL 9300 to (-40.42, 151.57, 135.08) mm, rotated rx -180 ry 0 rz 180 deg; joints [-52.881, -19.207, 99.128, 82.455, 53.547, -77.433]
  Call Extruder(4.34337)
  MoveL 9301 to (-40.47, 151.32, 135.08) mm, rotated rx 180 ry 0 rz 180 deg; joints [-52.862, -19.24, 99.15, 82.442, 53.53, -77.418]
  MoveL 9302 to (-40.47, 151.32, 135.08) mm, rotated rx 180 ry 0 rz 180 deg; joints [-52.862, -19.24, 99.15, 82.442, 53.53, -77.418]
  Call Extruder(4.47734)
  MoveL 9303 to (-40.52, 151.07, 135.08) mm, rotated rx 180 ry 0 rz 180 deg; joints [-52.843, -19.273, 99.173, 82.43, 53.513, -77.402]
  MoveL 9304 to (-40.52, 151.07, 135.08) mm, rotated rx 180 ry 0 rz 180 deg; joints [-52.843, -19.273, 99.173, 82.43, 53.513, -77.402]
  Call Extruder(4.61071)
  MoveL 9305 to (-40.56, 150.82, 135.08) mm, rotated rx 180 ry 0 rz 180 deg; joints [-52.824, -19.306, 99.196, 82.417, 53.496, -77.386]
  MoveL 9306 to (-40.56, 150.82, 135.08) mm, rotated rx 180 ry 0 rz 180 deg; joints [-52.824, -19.306, 99.196, 82.417, 53.496, -77.386]
  Call Extruder(4.77280)
  MoveL 9307 to (-40.61, 150.52, 135.08) mm, rotated rx 180 ry 0 rz 180 deg; joints [-52.799, -19.345, 99.223, 82.401, 53.473, -77.366]
  MoveL 9308 to (-40.61, 150.52, 135.08) mm, rotated rx 180 ry 0 rz 180 deg; joints [-52.799, -19.345, 99.223, 82.401, 53.473, -77.366]
  Call Extruder(4.93416)
  MoveL 9309 to (-40.66, 150.21, 135.08) mm, rotated rx 180 ry 0 rz 180 deg; joints [-52.775, -19.385, 99.25, 82.385, 53.451, -77.347]
  MoveL 9310 to (-40.66, 150.21, 135.08) mm, rotated rx 180 ry 0 rz 180 deg; joints [-52.775, -19.385, 99.25, 82.385, 53.451, -77.347]
  Call Extruder(5.09479)
  MoveL 9311 to (-40.71, 149.91, 135.08) mm, rotated rx 180 ry 0 rz 180 deg; joints [-52.75, -19.425, 99.277, 82.369, 53.428, -77.327]
  MoveL 9312 to (-40.71, 149.91, 135.08) mm, rotated rx 180 ry 0 rz 180 deg; joints [-52.75, -19.425, 99.277, 82.369, 53.428, -77.327]
  Call Extruder(5.25470)
  MoveL 9313 to (-40.76, 149.6, 135.08) mm, rotated rx 180 ry 0 rz -180 deg; joints [-52.725, -19.464, 99.304, 82.353, 53.405, -77.308]
  MoveL 9314 to (-40.76, 149.6, 135.08) mm, rotated rx 180 ry 0 rz -180 deg; joints [-52.725, -19.464, 99.304, 82.353, 53.405, -77.308]
  Call Extruder(5.41388)
  MoveL 9315 to (-40.81, 149.3, 135.08) mm, rotated rx 180 ry 0 rz 180 deg; joints [-52.7, -19.504, 99.331, 82.337, 53.383, -77.288]
  MoveL 9316 to (-40.81, 149.3, 135.08) mm, rotated rx 180 ry 0 rz 180 deg; joints [-52.7, -19.504, 99.331, 82.337, 53.383, -77.288]
  Call Extruder(5.57233)
  MoveL 9317 to (-40.86, 148.99, 135.08) mm, rotated rx -180 ry 0 rz 180 deg; joints [-52.675, -19.543, 99.358, 82.321, 53.36, -77.268]
  MoveL 9318 to (-40.86, 148.99, 135.08) mm, rotated rx -180 ry 0 rz 180 deg; joints [-52.675, -19.543, 99.358, 82.321, 53.36, -77.268]
  Call Extruder(5.77120)
  MoveL 9319 to (-40.9, 148.6, 135.08) mm, rotated rx 180 ry 0 rz -180 deg; joints [-52.641, -19.592, 99.391, 82.3, 53.329, -77.244]
  MoveL 9320 to (-40.9, 148.6, 135.08) mm, rotated rx 180 ry 0 rz -180 deg; joints [-52.641, -19.592, 99.391, 82.3, 53.329, -77.244]
  Call Extruder(5.96921)
  MoveL 9321 to (-40.95, 148.22, 135.08) mm, rotated rx 180 ry 0 rz 180 deg; joints [-52.607, -19.641, 99.424, 82.279, 53.298, -77.219]
  MoveL 9322 to (-40.95, 148.22, 135.08) mm, rotated rx 180 ry 0 rz 180 deg; joints [-52.607, -19.641, 99.424, 82.279, 53.298, -77.219]
  Call Extruder(6.16635)
  MoveL 9323 to (-40.99, 147.83, 135.08) mm, rotated rx 180 ry 0 rz 180 deg; joints [-52.573, -19.689, 99.457, 82.258, 53.267, -77.194]
  MoveL 9324 to (-40.99, 147.83, 135.08) mm, rotated rx 180 ry 0 rz 180 deg; joints [-52.573, -19.689, 99.457, 82.258, 53.267, -77.194]
  Call Extruder(6.36262)
  MoveL 9325 to (-41.04, 147.44, 135.08) mm, rotated rx 180 ry 0 rz 180 deg; joints [-52.539, -19.738, 99.49, 82.237, 53.236, -77.169]
  MoveL 9326 to (-41.04, 147.44, 135.08) mm, rotated rx 180 ry 0 rz 180 deg; joints [-52.539, -19.738, 99.49, 82.237, 53.236, -77.169]
  Call Extruder(6.60831)
  MoveL 9327 to (-41.09, 146.95, 135.08) mm, rotated rx -180 ry 0 rz 180 deg; joints [-52.494, -19.798, 99.531, 82.21, 53.195, -77.137]
  MoveL 9328 to (-41.09, 146.95, 135.08) mm, rotated rx -180 ry 0 rz 180 deg; joints [-52.494, -19.798, 99.531, 82.21, 53.195, -77.137]
  Call Extruder(6.90304)
  MoveL 9329 to (-41.13, 146.36, 135.08) mm, rotated rx -180 ry 0 rz 180 deg; joints [-52.439, -19.87, 99.579, 82.178, 53.144, -77.099]
  MoveL 9330 to (-41.13, 146.36, 135.08) mm, rotated rx -180 ry 0 rz 180 deg; joints [-52.439, -19.87, 99.579, 82.178, 53.144, -77.099]
  Call Extruder(7.19644)
  MoveL 9331 to (-41.18, 145.77, 135.08) mm, rotated rx 180 ry 0 rz 180 deg; joints [-52.383, -19.942, 99.628, 82.145, 53.093, -77.061]
  MoveL 9332 to (-41.18, 145.77, 135.08) mm, rotated rx 180 ry 0 rz 180 deg; joints [-52.383, -19.942, 99.628, 82.145, 53.093, -77.061]
  Call Extruder(7.62977)
  MoveL 9333 to (-41.23, 144.9, 135.08) mm, rotated rx -180 ry 0 rz 180 deg; joints [-52.297, -20.046, 99.698, 82.095, 53.014, -77.004]
  MoveL 9334 to (-41.23, 144.9, 135.08) mm, rotated rx -180 ry 0 rz 180 deg; joints [-52.297, -20.046, 99.698, 82.095, 53.014, -77.004]
  Call Extruder(8.20193)
  MoveL 9335 to (-41.27, 143.74, 135.08) mm, rotated rx -180 ry 0 rz -180 deg; joints [-52.18, -20.183, 99.79, 82.029, 52.906, -76.929]
  MoveL 9336 to (-41.27, 143.74, 135.08) mm, rotated rx -180 ry 0 rz -180 deg; joints [-52.18, -20.183, 99.79, 82.029, 52.906, -76.929]
  Call Extruder(8.62976)
  MoveL 9337 to (-41.29, 142.86, 135.08) mm, rotated rx -180 ry 0 rz 180 deg; joints [-52.09, -20.285, 99.858, 81.978, 52.823, -76.872]
  Call Extruder(50.62329)
  MoveL 9338 to (-41.29, 57.14, 135.08) mm, rotated rx 180 ry 0 rz 180 deg; joints [-40.759, -29.19, 105.156, 74.287, 42.705, -69.051]
  MoveL 9339 to (-41.29, 57.14, 135.08) mm, rotated rx 180 ry 0 rz 180 deg; joints [-40.759, -29.19, 105.156, 74.287, 42.705, -69.051]
  Call Extruder(51.33886)
  MoveL 9340 to (-41.25, 55.68, 135.08) mm, rotated rx 180 ry 0 rz -180 deg; joints [-40.517, -29.319, 105.223, 74.093, 42.496, -68.868]
  MoveL 9341 to (-41.25, 55.68, 135.08) mm, rotated rx 180 ry 0 rz -180 deg; joints [-40.517, -29.319, 105.223, 74.093, 42.496, -68.868]
  Call Extruder(51.91360)
  MoveL 9342 to (-41.2, 54.52, 135.08) mm, rotated rx 180 ry 0 rz 180 deg; joints [-40.32, -29.42, 105.275, 73.937, 42.326, -68.721]
  MoveL 9343 to (-41.2, 54.52, 135.08) mm, rotated rx 180 ry 0 rz 180 deg; joints [-40.32, -29.42, 105.275, 73.937, 42.326, -68.721]
  Call Extruder(52.20698)
  MoveL 9344 to (-41.15, 53.93, 135.08) mm, rotated rx 180 ry 0 rz 180 deg; joints [-40.217, -29.468, 105.3, 73.856, 42.236, -68.646]
  MoveL 9345 to (-41.15, 53.93, 135.08) mm, rotated rx 180 ry 0 rz 180 deg; joints [-40.217, -29.468, 105.3, 73.856, 42.236, -68.646]
  Call Extruder(52.50168)
  MoveL 9346 to (-41.11, 53.34, 135.08) mm, rotated rx 180 ry 0 rz 180 deg; joints [-40.114, -29.516, 105.325, 73.775, 42.147, -68.571]
  MoveL 9347 to (-41.11, 53.34, 135.08) mm, rotated rx 180 ry 0 rz 180 deg; joints [-40.114, -29.516, 105.325, 73.775, 42.147, -68.571]
  Call Extruder(52.79772)
  MoveL 9348 to (-41.06, 52.75, 135.08) mm, rotated rx -180 ry 0 rz 180 deg; joints [-40.01, -29.565, 105.35, 73.694, 42.057, -68.495]
  MoveL 9349 to (-41.06, 52.75, 135.08) mm, rotated rx -180 ry 0 rz 180 deg; joints [-40.01, -29.565, 105.35, 73.694, 42.057, -68.495]
  Call Extruder(52.99180)
  MoveL 9350 to (-41.02, 52.37, 135.08) mm, rotated rx 180 ry 0 rz 180 deg; joints [-39.94, -29.594, 105.365, 73.64, 41.996, -68.446]
  MoveL 9351 to (-41.02, 52.37, 135.08) mm, rotated rx 180 ry 0 rz 180 deg; joints [-39.94, -29.594, 105.365, 73.64, 41.996, -68.446]
  Call Extruder(53.18958)
  MoveL 9352 to (-40.97, 51.98, 135.08) mm, rotated rx 180 ry 0 rz 180 deg; joints [-39.869, -29.624, 105.381, 73.585, 41.934, -68.396]
  MoveL 9353 to (-40.97, 51.98, 135.08) mm, rotated rx 180 ry 0 rz 180 deg; joints [-39.869, -29.624, 105.381, 73.585, 41.934, -68.396]
  Call Extruder(53.38824)
  MoveL 9354 to (-40.93, 51.59, 135.08) mm, rotated rx 180 ry 0 rz 180 deg; joints [-39.798, -29.654, 105.396, 73.531, 41.872, -68.346]
  MoveL 9355 to (-40.93, 51.59, 135.08) mm, rotated rx 180 ry 0 rz 180 deg; joints [-39.798, -29.654, 105.396, 73.531, 41.872, -68.346]
  Call Extruder(53.58777)
  MoveL 9356 to (-40.88, 51.2, 135.08) mm, rotated rx 180 ry 0 rz 180 deg; joints [-39.727, -29.684, 105.411, 73.476, 41.81, -68.296]
  MoveL 9357 to (-40.88, 51.2, 135.08) mm, rotated rx 180 ry 0 rz 180 deg; joints [-39.727, -29.684, 105.411, 73.476, 41.81, -68.296]
  Call Extruder(53.76717)
  MoveL 9358 to (-40.83, 50.86, 135.08) mm, rotated rx 180 ry 0 rz 180 deg; joints [-39.663, -29.71, 105.425, 73.426, 41.754, -68.251]
  MoveL 9359 to (-40.83, 50.86, 135.08) mm, rotated rx 180 ry 0 rz 180 deg; joints [-39.663, -29.71, 105.425, 73.426, 41.754, -68.251]
  Call Extruder(53.92635)
  MoveL 9360 to (-40.78, 50.55, 135.08) mm, rotated rx 180 ry 0 rz 180 deg; joints [-39.605, -29.732, 105.436, 73.382, 41.704, -68.211]
  MoveL 9361 to (-40.78, 50.55, 135.08) mm, rotated rx 180 ry 0 rz 180 deg; joints [-39.605, -29.732, 105.436, 73.382, 41.704, -68.211]
  Call Extruder(54.08625)
  MoveL 9362 to (-40.74, 50.24, 135.08) mm, rotated rx 180 ry 0 rz 180 deg; joints [-39.547, -29.755, 105.447, 73.338, 41.653, -68.171]
  MoveL 9363 to (-40.74, 50.24, 135.08) mm, rotated rx 180 ry 0 rz 180 deg; joints [-39.547, -29.755, 105.447, 73.338, 41.653, -68.171]
  Call Extruder(54.24689)
  MoveL 9364 to (-40.69, 49.94, 135.08) mm, rotated rx 180 ry 0 rz -180 deg; joints [-39.489, -29.777, 105.458, 73.294, 41.602, -68.132]
  MoveL 9365 to (-40.69, 49.94, 135.08) mm, rotated rx 180 ry 0 rz -180 deg; joints [-39.489, -29.777, 105.458, 73.294, 41.602, -68.132]
  Call Extruder(54.40825)
  MoveL 9366 to (-40.64, 49.63, 135.08) mm, rotated rx 180 ry 0 rz 180 deg; joints [-39.431, -29.799, 105.47, 73.25, 41.552, -68.092]
  MoveL 9367 to (-40.64, 49.63, 135.08) mm, rotated rx 180 ry 0 rz 180 deg; joints [-39.431, -29.799, 105.47, 73.25, 41.552, -68.092]
  Call Extruder(54.57034)
  MoveL 9368 to (-40.59, 49.33, 135.08) mm, rotated rx -180 ry 0 rz 180 deg; joints [-39.373, -29.821, 105.481, 73.206, 41.501, -68.052]
  MoveL 9369 to (-40.59, 49.33, 135.08) mm, rotated rx -180 ry 0 rz 180 deg; joints [-39.373, -29.821, 105.481, 73.206, 41.501, -68.052]
  Call Extruder(54.71853)
  MoveL 9370 to (-40.54, 49.05, 135.08) mm, rotated rx 180 ry 0 rz 180 deg; joints [-39.32, -29.84, 105.491, 73.166, 41.454, -68.016]
  MoveL 9371 to (-40.54, 49.05, 135.08) mm, rotated rx 180 ry 0 rz 180 deg; joints [-39.32, -29.84, 105.491, 73.166, 41.454, -68.016]
  Call Extruder(54.85276)
  MoveL 9372 to (-40.49, 48.8, 135.08) mm, rotated rx 180 ry 0 rz 180 deg; joints [-39.271, -29.857, 105.499, 73.129, 41.411, -67.983]
  MoveL 9373 to (-40.49, 48.8, 135.08) mm, rotated rx 180 ry 0 rz 180 deg; joints [-39.271, -29.857, 105.499, 73.129, 41.411, -67.983]
  Call Extruder(54.98760)
  MoveL 9374 to (-40.44, 48.55, 135.08) mm, rotated rx 180 ry 0 rz 180 deg; joints [-39.222, -29.873, 105.508, 73.092, 41.369, -67.95]
  MoveL 9375 to (-40.44, 48.55, 135.08) mm, rotated rx 180 ry 0 rz 180 deg; joints [-39.222, -29.873, 105.508, 73.092, 41.369, -67.95]
  Call Extruder(55.12305)
  MoveL 9376 to (-40.39, 48.3, 135.08) mm, rotated rx 180 ry 0 rz 180 deg; joints [-39.174, -29.89, 105.516, 73.056, 41.326, -67.918]
  MoveL 9377 to (-40.39, 48.3, 135.08) mm, rotated rx 180 ry 0 rz 180 deg; joints [-39.174, -29.89, 105.516, 73.056, 41.326, -67.918]
  Call Extruder(55.25911)
  MoveL 9378 to (-40.34, 48.05, 135.08) mm, rotated rx 180 ry 0 rz 180 deg; joints [-39.125, -29.907, 105.525, 73.019, 41.283, -67.885]
  MoveL 9379 to (-40.34, 48.05, 135.08) mm, rotated rx 180 ry 0 rz 180 deg; joints [-39.125, -29.907, 105.525, 73.019, 41.283, -67.885]
  Call Extruder(55.39578)
  MoveL 9380 to (-40.29, 47.8, 135.08) mm, rotated rx -180 ry 0 rz -180 deg; joints [-39.076, -29.923, 105.533, 72.982, 41.24, -67.852]
  MoveL 9381 to (-40.29, 47.8, 135.08) mm, rotated rx -180 ry 0 rz -180 deg; joints [-39.076, -29.923, 105.533, 72.982, 41.24, -67.852]
  Call Extruder(55.53306)
  MoveL 9382 to (-40.24, 47.55, 135.08) mm, rotated rx 180 ry 0 rz 180 deg; joints [-39.027, -29.94, 105.542, 72.945, 41.197, -67.819]
  MoveL 9383 to (-40.24, 47.55, 135.08) mm, rotated rx 180 ry 0 rz 180 deg; joints [-39.027, -29.94, 105.542, 72.945, 41.197, -67.819]
  Call Extruder(55.65874)
  MoveL 9384 to (-40.2, 47.33, 135.08) mm, rotated rx 180 ry 0 rz 180 deg; joints [-38.982, -29.955, 105.549, 72.911, 41.158, -67.789]
  MoveL 9385 to (-40.2, 47.33, 135.08) mm, rotated rx 180 ry 0 rz 180 deg; joints [-38.982, -29.955, 105.549, 72.911, 41.158, -67.789]
  Call Extruder(55.77269)
  MoveL 9386 to (-40.15, 47.12, 135.08) mm, rotated rx 180 ry 0 rz 180 deg; joints [-38.941, -29.968, 105.556, 72.881, 41.122, -67.762]
  MoveL 9387 to (-40.15, 47.12, 135.08) mm, rotated rx 180 ry 0 rz 180 deg; joints [-38.941, -29.968, 105.556, 72.881, 41.122, -67.762]
  Call Extruder(55.88710)
  MoveL 9388 to (-40.11, 46.92, 135.08) mm, rotated rx 180 ry 0 rz 180 deg; joints [-38.9, -29.981, 105.562, 72.85, 41.086, -67.735]
  MoveL 9389 to (-40.11, 46.92, 135.08) mm, rotated rx 180 ry 0 rz 180 deg; joints [-38.9, -29.981, 105.562, 72.85, 41.086, -67.735]
  Call Extruder(56.00196)
  MoveL 9390 to (-40.06, 46.72, 135.08) mm, rotated rx -180 ry 0 rz 180 deg; joints [-38.859, -29.994, 105.569, 72.82, 41.05, -67.708]
  MoveL 9391 to (-40.06, 46.72, 135.08) mm, rotated rx -180 ry 0 rz 180 deg; joints [-38.859, -29.994, 105.569, 72.82, 41.05, -67.708]
  Call Extruder(56.11727)
  MoveL 9392 to (-40.02, 46.51, 135.08) mm, rotated rx 180 ry 0 rz 180 deg; joints [-38.819, -30.007, 105.576, 72.789, 41.014, -67.68]
  MoveL 9393 to (-40.02, 46.51, 135.08) mm, rotated rx 180 ry 0 rz 180 deg; joints [-38.819, -30.007, 105.576, 72.789, 41.014, -67.68]
  Call Extruder(56.24665)
  MoveL 9394 to (-39.95, 46.29, 135.08) mm, rotated rx -180 ry 0 rz 180 deg; joints [-38.771, -30.019, 105.582, 72.755, 40.972, -67.651]
  MoveL 9395 to (-39.95, 46.29, 135.08) mm, rotated rx -180 ry 0 rz 180 deg; joints [-38.771, -30.019, 105.582, 72.755, 40.972, -67.651]
  Call Extruder(56.37660)
  MoveL 9396 to (-39.88, 46.06, 135.08) mm, rotated rx -180 ry 0 rz 180 deg; joints [-38.724, -30.032, 105.588, 72.721, 40.93, -67.621]
  MoveL 9397 to (-39.88, 46.06, 135.08) mm, rotated rx -180 ry 0 rz 180 deg; joints [-38.724, -30.032, 105.588, 72.721, 40.93, -67.621]
  Call Extruder(56.50711)
  MoveL 9398 to (-39.82, 45.84, 135.08) mm, rotated rx -180 ry 0 rz 180 deg; joints [-38.677, -30.044, 105.594, 72.686, 40.888, -67.592]
  MoveL 9399 to (-39.82, 45.84, 135.08) mm, rotated rx -180 ry 0 rz 180 deg; joints [-38.677, -30.044, 105.594, 72.686, 40.888, -67.592]
  Call Extruder(56.63818)
  MoveL 9400 to (-39.75, 45.62, 135.08) mm, rotated rx -180 ry 0 rz -180 deg; joints [-38.629, -30.056, 105.6, 72.652, 40.846, -67.562]
  MoveL 9401 to (-39.75, 45.62, 135.08) mm, rotated rx -180 ry 0 rz -180 deg; joints [-38.629, -30.056, 105.6, 72.652, 40.846, -67.562]
  Call Extruder(56.75983)
  MoveL 9402 to (-39.68, 45.41, 135.08) mm, rotated rx 180 ry 0 rz 180 deg; joints [-38.585, -30.067, 105.606, 72.62, 40.807, -67.535]
  MoveL 9403 to (-39.68, 45.41, 135.08) mm, rotated rx 180 ry 0 rz 180 deg; joints [-38.585, -30.067, 105.606, 72.62, 40.807, -67.535]
  Call Extruder(56.87195)
  MoveL 9404 to (-39.62, 45.22, 135.08) mm, rotated rx 180 ry 0 rz -180 deg; joints [-38.544, -30.077, 105.611, 72.591, 40.771, -67.51]
  MoveL 9405 to (-39.62, 45.22, 135.08) mm, rotated rx 180 ry 0 rz -180 deg; joints [-38.544, -30.077, 105.611, 72.591, 40.771, -67.51]
  Call Extruder(56.98452)
  MoveL 9406 to (-39.56, 45.03, 135.08) mm, rotated rx 180 ry 0 rz 180 deg; joints [-38.504, -30.086, 105.616, 72.562, 40.735, -67.484]
  MoveL 9407 to (-39.56, 45.03, 135.08) mm, rotated rx 180 ry 0 rz 180 deg; joints [-38.504, -30.086, 105.616, 72.562, 40.735, -67.484]
  Call Extruder(57.09753)
  MoveL 9408 to (-39.5, 44.85, 135.08) mm, rotated rx -180 ry 0 rz -180 deg; joints [-38.463, -30.096, 105.621, 72.533, 40.699, -67.459]
  MoveL 9409 to (-39.5, 44.85, 135.08) mm, rotated rx -180 ry 0 rz -180 deg; joints [-38.463, -30.096, 105.621, 72.533, 40.699, -67.459]
  Call Extruder(57.21099)
  MoveL 9410 to (-39.44, 44.66, 135.08) mm, rotated rx 180 ry 0 rz 180 deg; joints [-38.422, -30.106, 105.625, 72.504, 40.662, -67.434]
  MoveL 9411 to (-39.44, 44.66, 135.08) mm, rotated rx 180 ry 0 rz 180 deg; joints [-38.422, -30.106, 105.625, 72.504, 40.662, -67.434]
  Call Extruder(57.35863)
  MoveL 9412 to (-39.35, 44.42, 135.08) mm, rotated rx 180 ry 0 rz -180 deg; joints [-38.369, -30.117, 105.631, 72.466, 40.614, -67.402]
  MoveL 9413 to (-39.35, 44.42, 135.08) mm, rotated rx 180 ry 0 rz -180 deg; joints [-38.369, -30.117, 105.631, 72.466, 40.614, -67.402]
  Call Extruder(57.54097)
  MoveL 9414 to (-39.23, 44.12, 135.08) mm, rotated rx 180 ry 0 rz 180 deg; joints [-38.302, -30.129, 105.637, 72.42, 40.555, -67.364]
  MoveL 9415 to (-39.23, 44.12, 135.08) mm, rotated rx 180 ry 0 rz 180 deg; joints [-38.302, -30.129, 105.637, 72.42, 40.555, -67.364]
  Call Extruder(57.72406)
  MoveL 9416 to (-39.11, 43.83, 135.08) mm, rotated rx -180 ry 0 rz 180 deg; joints [-38.236, -30.141, 105.643, 72.374, 40.495, -67.325]
  MoveL 9417 to (-39.11, 43.83, 135.08) mm, rotated rx -180 ry 0 rz 180 deg; joints [-38.236, -30.141, 105.643, 72.374, 40.495, -67.325]
  Call Extruder(57.88175)
  MoveL 9418 to (-39, 43.58, 135.08) mm, rotated rx 180 ry 0 rz 180 deg; joints [-38.178, -30.151, 105.648, 72.334, 40.444, -67.292]
  MoveL 9419 to (-39, 43.58, 135.08) mm, rotated rx 180 ry 0 rz 180 deg; joints [-38.178, -30.151, 105.648, 72.334, 40.444, -67.292]
  Call Extruder(58.04004)
  MoveL 9420 to (-38.89, 43.34, 135.08) mm, rotated rx 180 ry 0 rz 180 deg; joints [-38.121, -30.16, 105.653, 72.295, 40.392, -67.258]
  MoveL 9421 to (-38.89, 43.34, 135.08) mm, rotated rx 180 ry 0 rz 180 deg; joints [-38.121, -30.16, 105.653, 72.295, 40.392, -67.258]
  Call Extruder(58.22206)
  MoveL 9422 to (-38.75, 43.06, 135.08) mm, rotated rx 180 ry 0 rz 180 deg; joints [-38.054, -30.169, 105.657, 72.25, 40.332, -67.222]
  MoveL 9423 to (-38.75, 43.06, 135.08) mm, rotated rx 180 ry 0 rz 180 deg; joints [-38.054, -30.169, 105.657, 72.25, 40.332, -67.222]
  Call Extruder(58.42862)
  MoveL 9424 to (-38.57, 42.75, 135.08) mm, rotated rx 180 ry 0 rz 180 deg; joints [-37.977, -30.176, 105.661, 72.2, 40.262, -67.182]
  MoveL 9425 to (-38.57, 42.75, 135.08) mm, rotated rx 180 ry 0 rz 180 deg; joints [-37.977, -30.176, 105.661, 72.2, 40.262, -67.182]
  Call Extruder(58.63595)
  MoveL 9426 to (-38.4, 42.45, 135.08) mm, rotated rx 180 ry 0 rz 180 deg; joints [-37.901, -30.183, 105.664, 72.151, 40.193, -67.142]
  MoveL 9427 to (-38.4, 42.45, 135.08) mm, rotated rx 180 ry 0 rz 180 deg; joints [-37.901, -30.183, 105.664, 72.151, 40.193, -67.142]
  Call Extruder(58.84406)
  MoveL 9428 to (-38.22, 42.15, 135.08) mm, rotated rx 180 ry 0 rz 180 deg; joints [-37.825, -30.189, 105.668, 72.101, 40.124, -67.102]
  MoveL 9429 to (-38.22, 42.15, 135.08) mm, rotated rx 180 ry 0 rz 180 deg; joints [-37.825, -30.189, 105.668, 72.101, 40.124, -67.102]
  Call Extruder(58.96178)
  MoveL 9430 to (-38.12, 41.97, 135.08) mm, rotated rx 180 ry 0 rz 180 deg; joints [-37.782, -30.193, 105.669, 72.073, 40.085, -67.079]
  MoveL 9431 to (-38.12, 41.97, 135.08) mm, rotated rx 180 ry 0 rz 180 deg; joints [-37.782, -30.193, 105.669, 72.073, 40.085, -67.079]
  Call Extruder(59.29462)
  MoveL 9432 to (-37.8, 41.52, 135.08) mm, rotated rx 180 ry 0 rz 180 deg; joints [-37.659, -30.195, 105.671, 71.997, 39.972, -67.021]
  MoveL 9433 to (-37.8, 41.52, 135.08) mm, rotated rx 180 ry 0 rz 180 deg; joints [-37.659, -30.195, 105.671, 71.997, 39.972, -67.021]
  Call Extruder(59.62865)
  MoveL 9434 to (-37.47, 41.07, 135.08) mm, rotated rx -180 ry 0 rz 180 deg; joints [-37.537, -30.197, 105.672, 71.921, 39.86, -66.962]
  MoveL 9435 to (-37.47, 41.07, 135.08) mm, rotated rx -180 ry 0 rz 180 deg; joints [-37.537, -30.197, 105.672, 71.921, 39.86, -66.962]
  Call Extruder(59.79624)
  MoveL 9436 to (-37.3, 40.85, 135.08) mm, rotated rx 180 ry 0 rz -180 deg; joints [-37.475, -30.198, 105.672, 71.883, 39.803, -66.932]
  Call Extruder(60.62555)
  MoveL 9437 to (-36.39, 39.81, 135.08) mm, rotated rx -180 ry 0 rz 180 deg; joints [-37.173, -30.185, 105.665, 71.705, 39.523, -66.799]
  Call Extruder(61.25663)
  MoveL 9438 to (-35.6, 39.11, 135.08) mm, rotated rx 180 ry 0 rz 180 deg; joints [-36.947, -30.156, 105.651, 71.581, 39.311, -66.712]
  MoveL 9439 to (-35.6, 39.11, 135.08) mm, rotated rx 180 ry 0 rz 180 deg; joints [-36.947, -30.156, 105.651, 71.581, 39.311, -66.712]
  Call Extruder(61.45419)
  MoveL 9440 to (-35.35, 38.9, 135.08) mm, rotated rx -180 ry 0 rz 180 deg; joints [-36.876, -30.146, 105.646, 71.543, 39.244, -66.685]
  Call Extruder(61.78821)
  MoveL 9441 to (-34.9, 38.57, 135.08) mm, rotated rx 180 ry 0 rz 180 deg; joints [-36.759, -30.123, 105.634, 71.483, 39.133, -66.646]
  MoveL 9442 to (-34.9, 38.57, 135.08) mm, rotated rx 180 ry 0 rz 180 deg; joints [-36.759, -30.123, 105.634, 71.483, 39.133, -66.646]
  Call Extruder(62.12104)
  MoveL 9443 to (-34.45, 38.24, 135.08) mm, rotated rx -180 ry 0 rz -180 deg; joints [-36.642, -30.1, 105.622, 71.423, 39.023, -66.606]
  MoveL 9444 to (-34.45, 38.24, 135.08) mm, rotated rx -180 ry 0 rz -180 deg; joints [-36.642, -30.1, 105.622, 71.423, 39.023, -66.606]
  Call Extruder(62.30029)
  MoveL 9445 to (-34.21, 38.07, 135.08) mm, rotated rx 180 ry 0 rz 180 deg; joints [-36.579, -30.087, 105.616, 71.39, 38.963, -66.585]
  MoveL 9446 to (-34.21, 38.07, 135.08) mm, rotated rx 180 ry 0 rz 180 deg; joints [-36.579, -30.087, 105.616, 71.39, 38.963, -66.585]
  Call Extruder(62.50840)
  MoveL 9447 to (-33.9, 37.89, 135.08) mm, rotated rx -180 ry 0 rz 180 deg; joints [-36.509, -30.067, 105.606, 71.357, 38.895, -66.564]
  MoveL 9448 to (-33.9, 37.89, 135.08) mm, rotated rx -180 ry 0 rz 180 deg; joints [-36.509, -30.067, 105.606, 71.357, 38.895, -66.564]
  Call Extruder(62.71573)
  MoveL 9449 to (-33.6, 37.71, 135.08) mm, rotated rx 180 ry 0 rz -180 deg; joints [-36.439, -30.047, 105.596, 71.324, 38.827, -66.544]
  MoveL 9450 to (-33.6, 37.71, 135.08) mm, rotated rx 180 ry 0 rz -180 deg; joints [-36.439, -30.047, 105.596, 71.324, 38.827, -66.544]
  Call Extruder(62.92229)
  MoveL 9451 to (-33.29, 37.54, 135.08) mm, rotated rx 180 ry 0 rz 180 deg; joints [-36.368, -30.028, 105.586, 71.291, 38.76, -66.524]
  MoveL 9452 to (-33.29, 37.54, 135.08) mm, rotated rx 180 ry 0 rz 180 deg; joints [-36.368, -30.028, 105.586, 71.291, 38.76, -66.524]
  Call Extruder(63.12806)
  MoveL 9453 to (-32.99, 37.36, 135.08) mm, rotated rx 180 ry 0 rz 180 deg; joints [-36.298, -30.008, 105.576, 71.257, 38.692, -66.504]
  MoveL 9454 to (-32.99, 37.36, 135.08) mm, rotated rx 180 ry 0 rz 180 deg; joints [-36.298, -30.008, 105.576, 71.257, 38.692, -66.504]
  Call Extruder(63.28636)
  MoveL 9455 to (-32.74, 37.26, 135.08) mm, rotated rx 180 ry 0 rz 180 deg; joints [-36.247, -29.989, 105.566, 71.236, 38.642, -66.493]
  MoveL 9456 to (-32.74, 37.26, 135.08) mm, rotated rx 180 ry 0 rz 180 deg; joints [-36.247, -29.989, 105.566, 71.236, 38.642, -66.493]
  Call Extruder(63.44406)
  MoveL 9457 to (-32.49, 37.15, 135.08) mm, rotated rx 180 ry 0 rz 180 deg; joints [-36.196, -29.969, 105.556, 71.215, 38.592, -66.482]
  MoveL 9458 to (-32.49, 37.15, 135.08) mm, rotated rx 180 ry 0 rz 180 deg; joints [-36.196, -29.969, 105.556, 71.215, 38.592, -66.482]
  Call Extruder(63.61415)
  MoveL 9459 to (-32.22, 37.03, 135.08) mm, rotated rx 180 ry 0 rz 180 deg; joints [-36.141, -29.948, 105.546, 71.192, 38.539, -66.47]
  MoveL 9460 to (-32.22, 37.03, 135.08) mm, rotated rx 180 ry 0 rz 180 deg; joints [-36.141, -29.948, 105.546, 71.192, 38.539, -66.47]
  Call Extruder(63.79648)
  MoveL 9461 to (-31.93, 36.91, 135.08) mm, rotated rx 180 ry 0 rz 180 deg; joints [-36.082, -29.925, 105.534, 71.168, 38.481, -66.458]
  MoveL 9462 to (-31.93, 36.91, 135.08) mm, rotated rx 180 ry 0 rz 180 deg; joints [-36.082, -29.925, 105.534, 71.168, 38.481, -66.458]
  Call Extruder(63.97805)
  MoveL 9463 to (-31.64, 36.79, 135.08) mm, rotated rx 180 ry 0 rz 180 deg; joints [-36.023, -29.902, 105.522, 71.144, 38.424, -66.446]
  MoveL 9464 to (-31.64, 36.79, 135.08) mm, rotated rx 180 ry 0 rz 180 deg; joints [-36.023, -29.902, 105.522, 71.144, 38.424, -66.446]
  Call Extruder(64.09151)
  MoveL 9465 to (-31.45, 36.73, 135.08) mm, rotated rx 180 ry 0 rz 180 deg; joints [-35.989, -29.886, 105.514, 71.131, 38.389, -66.441]
  MoveL 9466 to (-31.45, 36.73, 135.08) mm, rotated rx 180 ry 0 rz 180 deg; joints [-35.989, -29.886, 105.514, 71.131, 38.389, -66.441]
  Call Extruder(64.20453)
  MoveL 9467 to (-31.26, 36.67, 135.08) mm, rotated rx 180 ry 0 rz 180 deg; joints [-35.954, -29.869, 105.506, 71.118, 38.354, -66.435]
  MoveL 9468 to (-31.26, 36.67, 135.08) mm, rotated rx 180 ry 0 rz 180 deg; joints [-35.954, -29.869, 105.506, 71.118, 38.354, -66.435]
  Call Extruder(64.31709)
  MoveL 9469 to (-31.07, 36.61, 135.08) mm, rotated rx 180 ry 0 rz 180 deg; joints [-35.919, -29.853, 105.497, 71.105, 38.32, -66.43]
  MoveL 9470 to (-31.07, 36.61, 135.08) mm, rotated rx 180 ry 0 rz 180 deg; joints [-35.919, -29.853, 105.497, 71.105, 38.32, -66.43]
  Call Extruder(64.42922)
  MoveL 9471 to (-30.88, 36.55, 135.08) mm, rotated rx 180 ry 0 rz 180 deg; joints [-35.884, -29.837, 105.489, 71.092, 38.285, -66.424]
  MoveL 9472 to (-30.88, 36.55, 135.08) mm, rotated rx 180 ry 0 rz 180 deg; joints [-35.884, -29.837, 105.489, 71.092, 38.285, -66.424]
  Call Extruder(64.54090)
  MoveL 9473 to (-30.69, 36.49, 135.08) mm, rotated rx 180 ry 0 rz 180 deg; joints [-35.849, -29.82, 105.481, 71.079, 38.251, -66.419]
  MoveL 9474 to (-30.69, 36.49, 135.08) mm, rotated rx 180 ry 0 rz 180 deg; joints [-35.849, -29.82, 105.481, 71.079, 38.251, -66.419]
  Call Extruder(64.67197)
  MoveL 9475 to (-30.47, 36.42, 135.08) mm, rotated rx 180 ry 0 rz 180 deg; joints [-35.809, -29.8, 105.471, 71.065, 38.211, -66.413]
  MoveL 9476 to (-30.47, 36.42, 135.08) mm, rotated rx 180 ry 0 rz 180 deg; joints [-35.809, -29.8, 105.471, 71.065, 38.211, -66.413]
  Call Extruder(64.80248)
